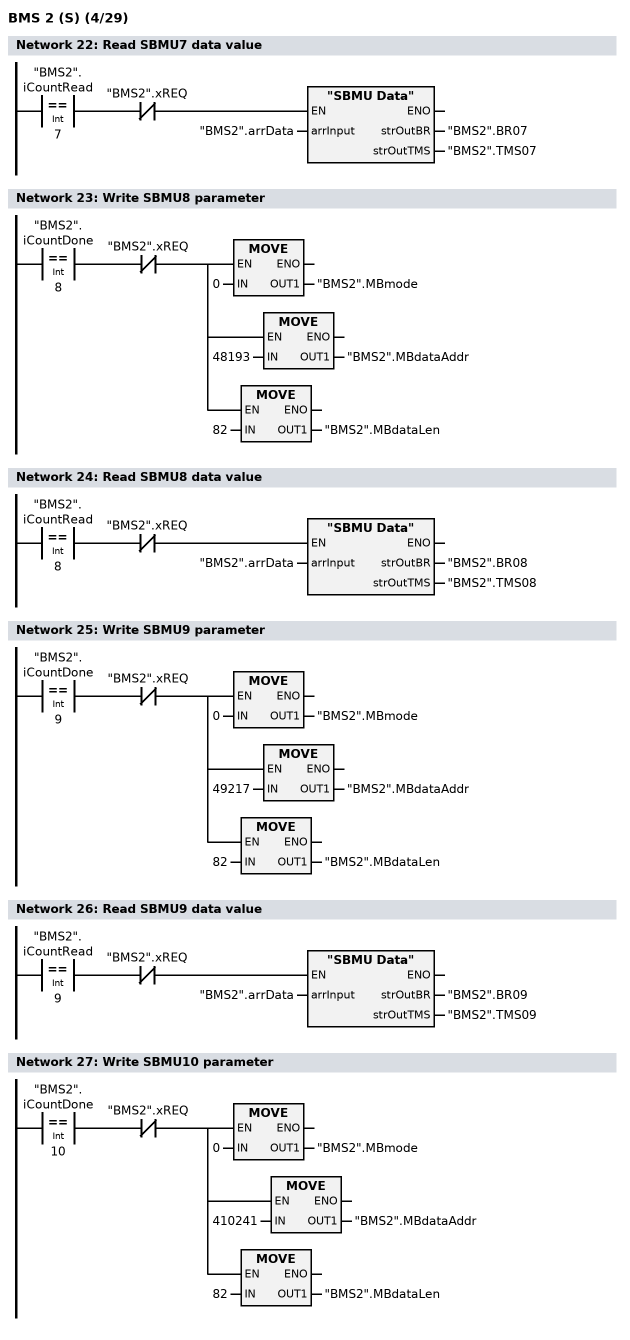
   RUNG wire#powerrail
      { S7_Templates := "SrcType := Int" } EQ_Contact(in1 := "BMS2".iCountRead, in2 := 7)
      I_Contact( "BMS2".xREQ )
      "SBMU Data"(arrInput := "BMS2".arrData, strOutBR => "BMS2".BR07, strOutTMS => "BMS2".TMS07)
   END_RUNG
   // the same network as SCL:
   IF ("BMS2".iCountRead = 7) AND NOT "BMS2".xREQ THEN
       "SBMU Data"(arrInput := "BMS2".arrData, strOutBR => "BMS2".BR07, strOutTMS => "BMS2".TMS07);
   END_IF;
END_REGION

REGION Network 23: Write SBMU8 parameter
   RUNG wire#powerrail
      { S7_Templates := "SrcType := Int" } EQ_Contact(in1 := "BMS2".iCountDone, in2 := 8)
      I_Contact( "BMS2".xREQ )
      wire#w1
      Move(in := 0, out1 => "BMS2".MBmode)
   END_RUNG
   RUNG wire#w1
      Move(in := 48193, out1 => "BMS2".MBdataAddr)
   END_RUNG
   RUNG wire#w1
      Move(in := 82, out1 => "BMS2".MBdataLen)
   END_RUNG
   // the same network as SCL:
   IF ("BMS2".iCountDone = 8) AND NOT "BMS2".xREQ THEN
       "BMS2".MBmode := 0;
       "BMS2".MBdataAddr := 48193;
       "BMS2".MBdataLen := 82;
   END_IF;
END_REGION

REGION Network 24: Read SBMU8 data value
   RUNG wire#powerrail
      { S7_Templates := "SrcType := Int" } EQ_Contact(in1 := "BMS2".iCountRead, in2 := 8)
      I_Contact( "BMS2".xREQ )
      "SBMU Data"(arrInput := "BMS2".arrData, strOutBR => "BMS2".BR08, strOutTMS => "BMS2".TMS08)
   END_RUNG
   // the same network as SCL:
   IF ("BMS2".iCountRead = 8) AND NOT "BMS2".xREQ THEN
       "SBMU Data"(arrInput := "BMS2".arrData, strOutBR => "BMS2".BR08, strOutTMS => "BMS2".TMS08);
   END_IF;
END_REGION

REGION Network 25: Write SBMU9 parameter
   RUNG wire#powerrail
      { S7_Templates := "SrcType := Int" } EQ_Contact(in1 := "BMS2".iCountDone, in2 := 9)
      I_Contact( "BMS2".xREQ )
      wire#w1
      Move(in := 0, out1 => "BMS2".MBmode)
   END_RUNG
   RUNG wire#w1
      Move(in := 49217, out1 => "BMS2".MBdataAddr)
   END_RUNG
   RUNG wire#w1
      Move(in := 82, out1 => "BMS2".MBdataLen)
   END_RUNG
   // the same network as SCL:
   IF ("BMS2".iCountDone = 9) AND NOT "BMS2".xREQ THEN
       "BMS2".MBmode := 0;
       "BMS2".MBdataAddr := 49217;
       "BMS2".MBdataLen := 82;
   END_IF;
END_REGION

REGION Network 26: Read SBMU9 data value
   RUNG wire#powerrail
      { S7_Templates := "SrcType := Int" } EQ_Contact(in1 := "BMS2".iCountRead, in2 := 9)
      I_Contact( "BMS2".xREQ )
      "SBMU Data"(arrInput := "BMS2".arrData, strOutBR => "BMS2".BR09, strOutTMS => "BMS2".TMS09)
   END_RUNG
   // the same network as SCL:
   IF ("BMS2".iCountRead = 9) AND NOT "BMS2".xREQ THEN
       "SBMU Data"(arrInput := "BMS2".arrData, strOutBR => "BMS2".BR09, strOutTMS => "BMS2".TMS09);
   END_IF;
END_REGION

REGION Network 27: Write SBMU10 parameter
   RUNG wire#powerrail
      { S7_Templates := "SrcType := Int" } EQ_Contact(in1 := "BMS2".iCountDone, in2 := 10)
      I_Contact( "BMS2".xREQ )
      wire#w1
      Move(in := 0, out1 => "BMS2".MBmode)
   END_RUNG
   RUNG wire#w1
      Move(in := 410241, out1 => "BMS2".MBdataAddr)
   END_RUNG
   RUNG wire#w1
      Move(in := 82, out1 => "BMS2".MBdataLen)
   END_RUNG
   // the same network as SCL:
   IF ("BMS2".iCountDone = 10) AND NOT "BMS2".xREQ THEN
       "BMS2".MBmode := 0;
       "BMS2".MBdataAddr := 410241;
       "BMS2".MBdataLen := 82;
   END_IF;
END_REGION

REGION Network 28: Read SBMU10 data value
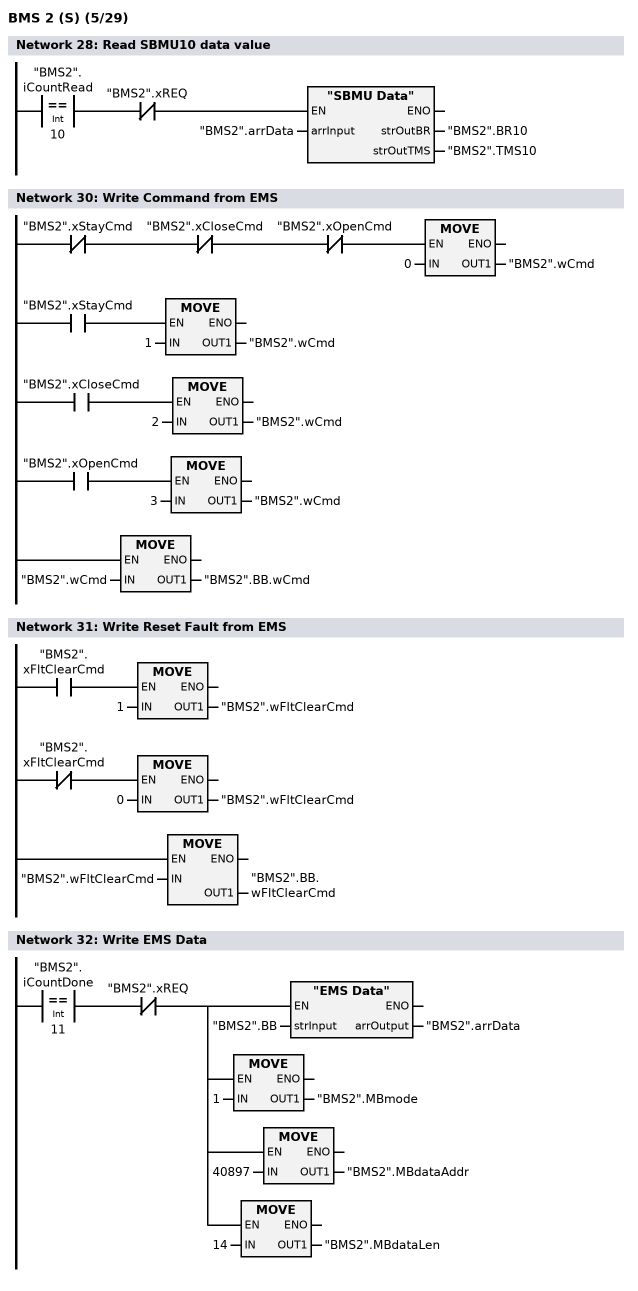
   RUNG wire#powerrail
      { S7_Templates := "SrcType := Int" } EQ_Contact(in1 := "BMS2".iCountRead, in2 := 10)
      I_Contact( "BMS2".xREQ )
      "SBMU Data"(arrInput := "BMS2".arrData, strOutBR => "BMS2".BR10, strOutTMS => "BMS2".TMS10)
   END_RUNG
   // the same network as SCL:
   IF ("BMS2".iCountRead = 10) AND NOT "BMS2".xREQ THEN
       "SBMU Data"(arrInput := "BMS2".arrData, strOutBR => "BMS2".BR10, strOutTMS => "BMS2".TMS10);
   END_IF;
END_REGION

REGION Network 30: Write Command from EMS
   RUNG wire#powerrail
      I_Contact( "BMS2".xStayCmd )
      I_Contact( "BMS2".xCloseCmd )
      I_Contact( "BMS2".xOpenCmd )
      Move(in := 0, out1 => "BMS2".wCmd)
   END_RUNG
   RUNG wire#powerrail
      Contact( "BMS2".xStayCmd )
      Move(in := 1, out1 => "BMS2".wCmd)
   END_RUNG
   RUNG wire#powerrail
      Contact( "BMS2".xCloseCmd )
      Move(in := 2, out1 => "BMS2".wCmd)
   END_RUNG
   RUNG wire#powerrail
      Contact( "BMS2".xOpenCmd )
      Move(in := 3, out1 => "BMS2".wCmd)
   END_RUNG
   RUNG wire#powerrail
      Move(in := "BMS2".wCmd, out1 => "BMS2".BB.wCmd)
   END_RUNG
   // the same network as SCL:
   IF NOT "BMS2".xStayCmd AND NOT "BMS2".xCloseCmd AND NOT "BMS2".xOpenCmd THEN "BMS2".wCmd := 0; END_IF;
   IF "BMS2".xStayCmd THEN "BMS2".wCmd := 1; END_IF;
   IF "BMS2".xCloseCmd THEN "BMS2".wCmd := 2; END_IF;
   IF "BMS2".xOpenCmd THEN "BMS2".wCmd := 3; END_IF;
   "BMS2".BB.wCmd := "BMS2".wCmd;
END_REGION

REGION Network 31: Write Reset Fault from EMS
   RUNG wire#powerrail
      Contact( "BMS2".xFltClearCmd )
      Move(in := 1, out1 => "BMS2".wFltClearCmd)
   END_RUNG
   RUNG wire#powerrail
      I_Contact( "BMS2".xFltClearCmd )
      Move(in := 0, out1 => "BMS2".wFltClearCmd)
   END_RUNG
   RUNG wire#powerrail
      Move(in := "BMS2".wFltClearCmd, out1 => "BMS2".BB.wFltClearCmd)
   END_RUNG
   // the same network as SCL:
   IF "BMS2".xFltClearCmd THEN "BMS2".wFltClearCmd := 1; END_IF;
   IF NOT "BMS2".xFltClearCmd THEN "BMS2".wFltClearCmd := 0; END_IF;
   "BMS2".BB.wFltClearCmd := "BMS2".wFltClearCmd;
END_REGION

REGION Network 32: Write EMS Data
   RUNG wire#powerrail
      { S7_Templates := "SrcType := Int" } EQ_Contact(in1 := "BMS2".iCountDone, in2 := 11)
      I_Contact( "BMS2".xREQ )
      wire#w1
      "EMS Data"(strInput := "BMS2".BB, arrOutput => "BMS2".arrData)
   END_RUNG
   RUNG wire#w1
      Move(in := 1, out1 => "BMS2".MBmode)
   END_RUNG
   RUNG wire#w1
      Move(in := 40897, out1 => "BMS2".MBdataAddr)
   END_RUNG
   RUNG wire#w1
      Move(in := 14, out1 => "BMS2".MBdataLen)
   END_RUNG
   // the same network as SCL:
   #_w1 := ("BMS2".iCountDone = 11) AND NOT "BMS2".xREQ;
   IF #_w1 THEN
       "EMS Data"(strInput := "BMS2".BB, arrOutput => "BMS2".arrData);
       "BMS2".MBmode := 1;
       "BMS2".MBdataAddr := 40897;
       "BMS2".MBdataLen := 14;
   END_IF;
END_REGION

REGION Network 34: Fault Modbus Communication
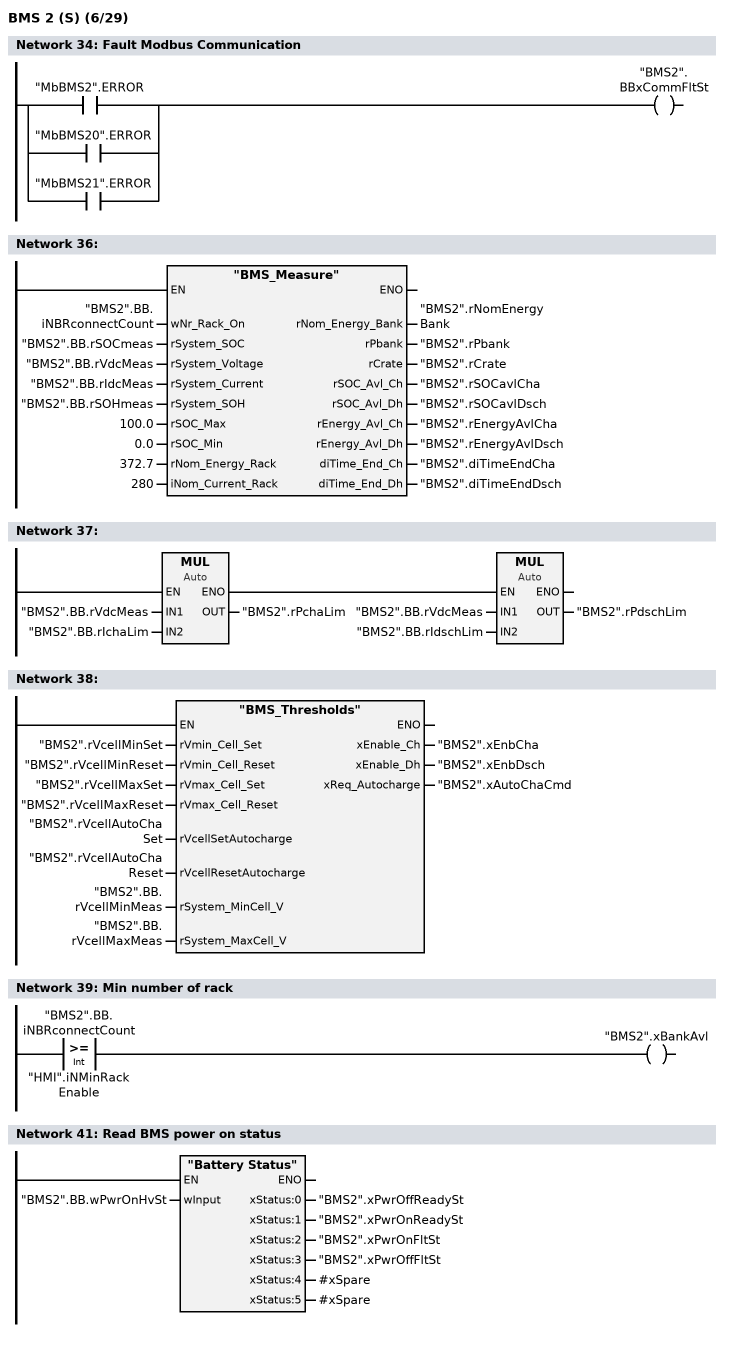
   RUNG wire#powerrail
      Contact( "MbBMS2".ERROR )
      wire#w1
      Coil( "BMS2".BBxCommFltSt )
   END_RUNG
   RUNG wire#powerrail
      Contact( "MbBMS20".ERROR )
   END_RUNG wire#w1
   RUNG wire#powerrail
      Contact( "MbBMS21".ERROR )
   END_RUNG wire#w1
   // the same network as SCL:
   "BMS2".BBxCommFltSt := "MbBMS2".ERROR OR "MbBMS20".ERROR OR "MbBMS21".ERROR;
END_REGION

REGION Network 36
   RUNG wire#powerrail
      "BMS_Measure"(wNr_Rack_On := "BMS2".BB.iNBRconnectCount, rSystem_SOC := "BMS2".BB.rSOCmeas, rSystem_Voltage := "BMS2".BB.rVdcMeas, rSystem_Current := "BMS2".BB.rIdcMeas, rSystem_SOH := "BMS2".BB.rSOHmeas, rSOC_Max := 100.0, rSOC_Min := 0.0, rNom_Energy_Rack := 372.7, iNom_Current_Rack := 280, rNom_Energy_Bank => "BMS2".rNomEnergyBank, rPbank => "BMS2".rPbank, rCrate => "BMS2".rCrate, rSOC_Avl_Ch => "BMS2".rSOCavlCha, rSOC_Avl_Dh => "BMS2".rSOCavlDsch, rEnergy_Avl_Ch => "BMS2".rEnergyAvlCha, rEnergy_Avl_Dh => "BMS2".rEnergyAvlDsch, diTime_End_Ch => "BMS2".diTimeEndCha, diTime_End_Dh => "BMS2".diTimeEndDsch)
   END_RUNG
   // the same network as SCL:
   "BMS_Measure"(wNr_Rack_On := "BMS2".BB.iNBRconnectCount,
                 rSystem_SOC := "BMS2".BB.rSOCmeas,
                 rSystem_Voltage := "BMS2".BB.rVdcMeas,
                 rSystem_Current := "BMS2".BB.rIdcMeas,
                 rSystem_SOH := "BMS2".BB.rSOHmeas,
                 rSOC_Max := 100.0,
                 rSOC_Min := 0.0,
                 rNom_Energy_Rack := 372.7,
                 iNom_Current_Rack := 280,
                 rNom_Energy_Bank => "BMS2".rNomEnergyBank,
                 rPbank => "BMS2".rPbank,
                 rCrate => "BMS2".rCrate,
                 rSOC_Avl_Ch => "BMS2".rSOCavlCha,
                 rSOC_Avl_Dh => "BMS2".rSOCavlDsch,
                 rEnergy_Avl_Ch => "BMS2".rEnergyAvlCha,
                 rEnergy_Avl_Dh => "BMS2".rEnergyAvlDsch,
                 diTime_End_Ch => "BMS2".diTimeEndCha,
                 diTime_End_Dh => "BMS2".diTimeEndDsch);
END_REGION

REGION Network 37
   RUNG wire#powerrail
      Mul(in1 := "BMS2".BB.rVdcMeas, in2 := "BMS2".BB.rIchaLim, out => "BMS2".rPchaLim)
      Mul(in1 := "BMS2".BB.rVdcMeas, in2 := "BMS2".BB.rIdschLim, out => "BMS2".rPdschLim)
   END_RUNG
   // the same network as SCL:
   "BMS2".rPchaLim := "BMS2".BB.rVdcMeas * "BMS2".BB.rIchaLim;
   "BMS2".rPdschLim := "BMS2".BB.rVdcMeas * "BMS2".BB.rIdschLim;
END_REGION

REGION Network 38
   RUNG wire#powerrail
      "BMS_Thresholds"(rVmin_Cell_Set := "BMS2".rVcellMinSet, rVmin_Cell_Reset := "BMS2".rVcellMinReset, rVmax_Cell_Set := "BMS2".rVcellMaxSet, rVmax_Cell_Reset := "BMS2".rVcellMaxReset, rVcellSetAutocharge := "BMS2".rVcellAutoChaSet, rVcellResetAutocharge := "BMS2".rVcellAutoChaReset, rSystem_MinCell_V := "BMS2".BB.rVcellMinMeas, rSystem_MaxCell_V := "BMS2".BB.rVcellMaxMeas, xEnable_Ch => "BMS2".xEnbCha, xEnable_Dh => "BMS2".xEnbDsch, xReq_Autocharge => "BMS2".xAutoChaCmd)
   END_RUNG
   // the same network as SCL:
   "BMS_Thresholds"(rVmin_Cell_Set := "BMS2".rVcellMinSet,
                    rVmin_Cell_Reset := "BMS2".rVcellMinReset,
                    rVmax_Cell_Set := "BMS2".rVcellMaxSet,
                    rVmax_Cell_Reset := "BMS2".rVcellMaxReset,
                    rVcellSetAutocharge := "BMS2".rVcellAutoChaSet,
                    rVcellResetAutocharge := "BMS2".rVcellAutoChaReset,
                    rSystem_MinCell_V := "BMS2".BB.rVcellMinMeas,
                    rSystem_MaxCell_V := "BMS2".BB.rVcellMaxMeas,
                    xEnable_Ch => "BMS2".xEnbCha,
                    xEnable_Dh => "BMS2".xEnbDsch,
                    xReq_Autocharge => "BMS2".xAutoChaCmd);
END_REGION

REGION Network 39: Min number of rack
   RUNG wire#powerrail
      { S7_Templates := "SrcType := Int" } GE_Contact(in1 := "BMS2".BB.iNBRconnectCount, in2 := "HMI".iNMinRackEnable)
      Coil( "BMS2".xBankAvl )
   END_RUNG
   // the same network as SCL:
   "BMS2".xBankAvl := "BMS2".BB.iNBRconnectCount >= "HMI".iNMinRackEnable;
END_REGION

REGION Network 41: Read BMS power on status
   RUNG wire#powerrail
      "Battery Status"(wInput := "BMS2".BB.wPwrOnHvSt, "xStatus:0" => "BMS2".xPwrOffReadySt, "xStatus:1" => "BMS2".xPwrOnReadySt, "xStatus:2" => "BMS2".xPwrOnFltSt, "xStatus:3" => "BMS2".xPwrOffFltSt, "xStatus:4" => #xSpare, "xStatus:5" => #xSpare)
   END_RUNG
   // the same network as SCL:
   "Battery Status"(wInput := "BMS2".BB.wPwrOnHvSt,
                    "xStatus:0" => "BMS2".xPwrOffReadySt,
                    "xStatus:1" => "BMS2".xPwrOnReadySt,
                    "xStatus:2" => "BMS2".xPwrOnFltSt,
                    "xStatus:3" => "BMS2".xPwrOffFltSt,
                    "xStatus:4" => #xSpare,
                    "xStatus:5" => #xSpare);
END_REGION

REGION Network 42: Read BMS status
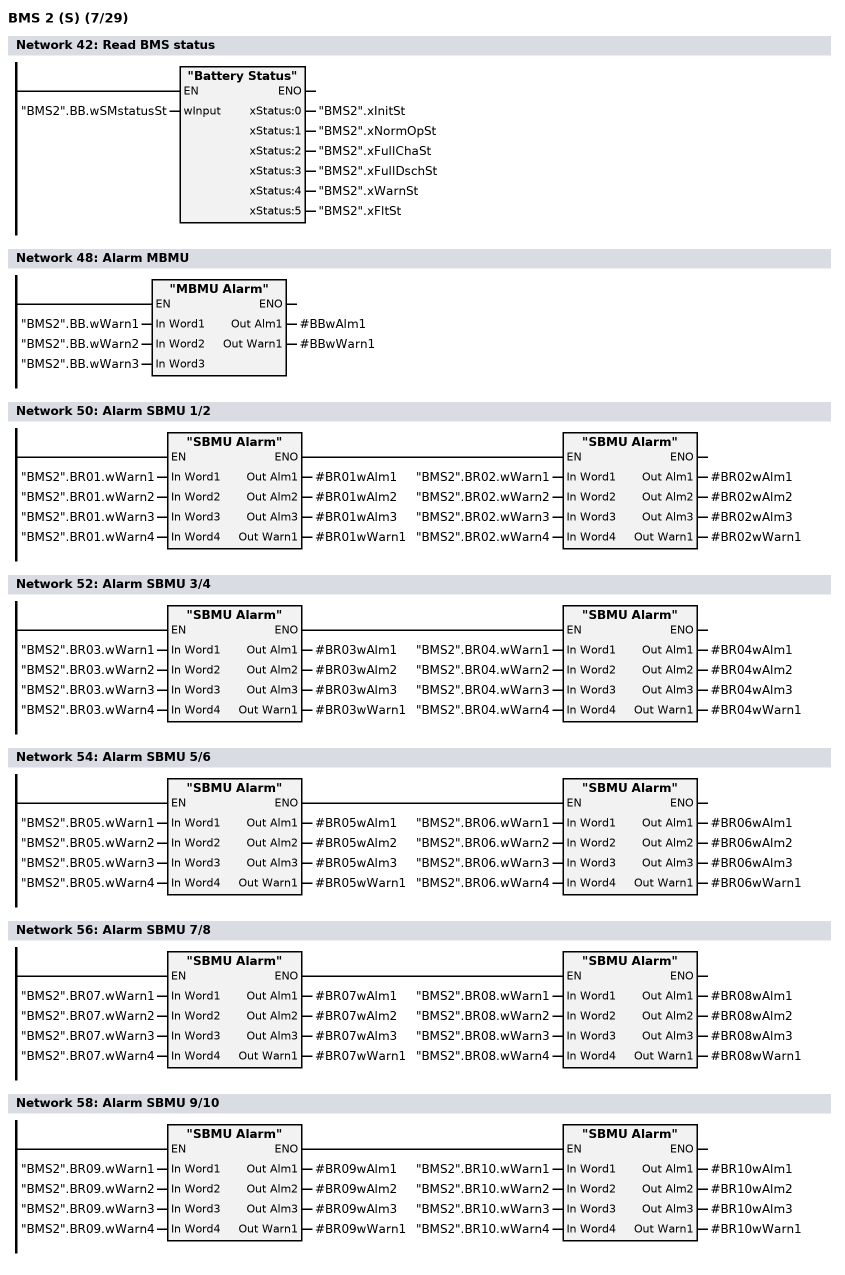
   RUNG wire#powerrail
      "Battery Status"(wInput := "BMS2".BB.wSMstatusSt, "xStatus:0" => "BMS2".xInitSt, "xStatus:1" => "BMS2".xNormOpSt, "xStatus:2" => "BMS2".xFullChaSt, "xStatus:3" => "BMS2".xFullDschSt, "xStatus:4" => "BMS2".xWarnSt, "xStatus:5" => "BMS2".xFltSt)
   END_RUNG
   // the same network as SCL:
   "Battery Status"(wInput := "BMS2".BB.wSMstatusSt,
                    "xStatus:0" => "BMS2".xInitSt,
                    "xStatus:1" => "BMS2".xNormOpSt,
                    "xStatus:2" => "BMS2".xFullChaSt,
                    "xStatus:3" => "BMS2".xFullDschSt,
                    "xStatus:4" => "BMS2".xWarnSt,
                    "xStatus:5" => "BMS2".xFltSt);
END_REGION

REGION Network 44 (SCL): Rack Fault Status
   "BMS2".wRackFlt.%X0 := "BMS2".BR01xFltSt;
   "BMS2".wRackFlt.%X1 := "BMS2".BR02xFltSt;
   "BMS2".wRackFlt.%X2 := "BMS2".BR03xFltSt;
   "BMS2".wRackFlt.%X3 := "BMS2".BR04xFltSt;
   "BMS2".wRackFlt.%X4 := "BMS2".BR05xFltSt;
   "BMS2".wRackFlt.%X5 := "BMS2".BR06xFltSt;
   "BMS2".wRackFlt.%X6 := "BMS2".BR07xFltSt;
   "BMS2".wRackFlt.%X7 := "BMS2".BR08xFltSt;
   "BMS2".wRackFlt.%X8 := "BMS2".BR09xFltSt;
   "BMS2".wRackFlt.%X9 := "BMS2".BR10xFltSt;
END_REGION

REGION Network 45 (SCL): Rack On Status
   "BMS2".wRackOn.%X0 := "BMS2".BR01.xKposSt;
   "BMS2".wRackOn.%X1 := "BMS2".BR02.xKposSt;
   "BMS2".wRackOn.%X2 := "BMS2".BR03.xKposSt;
   "BMS2".wRackOn.%X3 := "BMS2".BR04.xKposSt;
   "BMS2".wRackOn.%X4 := "BMS2".BR05.xKposSt;
   "BMS2".wRackOn.%X5 := "BMS2".BR06.xKposSt;
   "BMS2".wRackOn.%X6 := "BMS2".BR07.xKposSt;
   "BMS2".wRackOn.%X7 := "BMS2".BR08.xKposSt;
   "BMS2".wRackOn.%X8 := "BMS2".BR09.xKposSt;
   "BMS2".wRackOn.%X9 := "BMS2".BR10.xKposSt;
END_REGION

REGION Network 46 (SCL): Status Switch Gear
   IF
       NOT "BMS2".BR01wAlm2.%X12 OR
       NOT "BMS2".BR02wAlm2.%X12 OR
       NOT "BMS2".BR03wAlm2.%X12 OR
       NOT "BMS2".BR04wAlm2.%X12 OR
       NOT "BMS2".BR05wAlm2.%X12 OR
       NOT "BMS2".BR06wAlm2.%X12 OR
       NOT "BMS2".BR07wAlm2.%X12 OR
       NOT "BMS2".BR08wAlm2.%X12 OR
       NOT "BMS2".BR09wAlm2.%X12 OR
       NOT "BMS2".BR10wAlm2.%X12 THEN

       "BMS2".xSwitchGearSt := True;
   ELSE
       "BMS2".xSwitchGearSt := False;
   END_IF;
END_REGION

REGION Network 48: Alarm MBMU
   RUNG wire#powerrail
      "MBMU Alarm"("In Word1" := "BMS2".BB.wWarn1, "In Word2" := "BMS2".BB.wWarn2, "In Word3" := "BMS2".BB.wWarn3, "Out Alm1" => #BBwAlm1, "Out Warn1" => #BBwWarn1)
   END_RUNG
   // the same network as SCL:
   "MBMU Alarm"("In Word1" := "BMS2".BB.wWarn1,
                "In Word2" := "BMS2".BB.wWarn2,
                "In Word3" := "BMS2".BB.wWarn3,
                "Out Alm1" => #BBwAlm1,
                "Out Warn1" => #BBwWarn1);
END_REGION

REGION Network 49 (SCL): Alarm MBMU to HMI
   IF "HMI".xBB2AlmDisable OR"HMI".xPEMSAlmDisable OR"HMI".xPIAlmDisable
   THEN
       "BMS2".BBwAlm1 := 0;
       "BMS2".BBwWarn1 := 0;
   ELSE
       "BMS2".BBwAlm1 := #BBwAlm1;
       "BMS2".BBwWarn1 := #BBwWarn1;
   END_IF;
END_REGION

REGION Network 50: Alarm SBMU 1/2
   RUNG wire#powerrail
      "SBMU Alarm"("In Word1" := "BMS2".BR01.wWarn1, "In Word2" := "BMS2".BR01.wWarn2, "In Word3" := "BMS2".BR01.wWarn3, "In Word4" := "BMS2".BR01.wWarn4, "Out Alm1" => #BR01wAlm1, "Out Alm2" => #BR01wAlm2, "Out Alm3" => #BR01wAlm3, "Out Warn1" => #BR01wWarn1)
      "SBMU Alarm"("In Word1" := "BMS2".BR02.wWarn1, "In Word2" := "BMS2".BR02.wWarn2, "In Word3" := "BMS2".BR02.wWarn3, "In Word4" := "BMS2".BR02.wWarn4, "Out Alm1" => #BR02wAlm1, "Out Alm2" => #BR02wAlm2, "Out Alm3" => #BR02wAlm3, "Out Warn1" => #BR02wWarn1)
   END_RUNG
   // the same network as SCL:
   "SBMU Alarm"("In Word1" := "BMS2".BR01.wWarn1,
                "In Word2" := "BMS2".BR01.wWarn2,
                "In Word3" := "BMS2".BR01.wWarn3,
                "In Word4" := "BMS2".BR01.wWarn4,
                "Out Alm1" => #BR01wAlm1,
                "Out Alm2" => #BR01wAlm2,
                "Out Alm3" => #BR01wAlm3,
                "Out Warn1" => #BR01wWarn1,
                ENO => #_w1);
   IF #_w1 THEN
       "SBMU Alarm"("In Word1" := "BMS2".BR02.wWarn1,
                    "In Word2" := "BMS2".BR02.wWarn2,
                    "In Word3" := "BMS2".BR02.wWarn3,
                    "In Word4" := "BMS2".BR02.wWarn4,
                    "Out Alm1" => #BR02wAlm1,
                    "Out Alm2" => #BR02wAlm2,
                    "Out Alm3" => #BR02wAlm3,
                    "Out Warn1" => #BR02wWarn1);
   END_IF;
END_REGION

REGION Network 51 (SCL): Alarm SBMU 1/2 to HMI
   IF "HMI".xBB2BR1AlmDisable OR "HMI".xBB2AlmDisable OR "HMI".xPEMSAlmDisable OR "HMI".xPIAlmDisable
   THEN
       "BMS2".BR01wAlm1 := 0;
       "BMS2".BR01wAlm2 := 0;
       "BMS2".BR01wAlm3 := 0;
       "BMS2".BR01wWarn1 := 0;
   ELSE
       "BMS2".BR01wAlm1 := #BR01wAlm1;
       "BMS2".BR01wAlm2 := #BR01wAlm2;
       "BMS2".BR01wAlm3 := #BR01wAlm3;
       "BMS2".BR01wWarn1 := #BR01wWarn1;
   END_IF;

   IF "HMI".xBB2BR2AlmDisable OR "HMI".xBB2AlmDisable OR "HMI".xPEMSAlmDisable OR "HMI".xPIAlmDisable
   THEN
       "BMS2".BR02wAlm1 := 0;
       "BMS2".BR02wAlm2 := 0;
       "BMS2".BR02wAlm3 := 0;
       "BMS2".BR02wWarn1 := 0;
   ELSE
       "BMS2".BR02wAlm1 := #BR02wAlm1;
       "BMS2".BR02wAlm2 := #BR02wAlm2;
       "BMS2".BR02wAlm3 := #BR02wAlm3;
       "BMS2".BR02wWarn1 := #BR02wWarn1;
   END_IF;
END_REGION

REGION Network 52: Alarm SBMU 3/4
   RUNG wire#powerrail
      "SBMU Alarm"("In Word1" := "BMS2".BR03.wWarn1, "In Word2" := "BMS2".BR03.wWarn2, "In Word3" := "BMS2".BR03.wWarn3, "In Word4" := "BMS2".BR03.wWarn4, "Out Alm1" => #BR03wAlm1, "Out Alm2" => #BR03wAlm2, "Out Alm3" => #BR03wAlm3, "Out Warn1" => #BR03wWarn1)
      "SBMU Alarm"("In Word1" := "BMS2".BR04.wWarn1, "In Word2" := "BMS2".BR04.wWarn2, "In Word3" := "BMS2".BR04.wWarn3, "In Word4" := "BMS2".BR04.wWarn4, "Out Alm1" => #BR04wAlm1, "Out Alm2" => #BR04wAlm2, "Out Alm3" => #BR04wAlm3, "Out Warn1" => #BR04wWarn1)
   END_RUNG
   // the same network as SCL:
   "SBMU Alarm"("In Word1" := "BMS2".BR03.wWarn1,
                "In Word2" := "BMS2".BR03.wWarn2,
                "In Word3" := "BMS2".BR03.wWarn3,
                "In Word4" := "BMS2".BR03.wWarn4,
                "Out Alm1" => #BR03wAlm1,
                "Out Alm2" => #BR03wAlm2,
                "Out Alm3" => #BR03wAlm3,
                "Out Warn1" => #BR03wWarn1,
                ENO => #_w1);
   IF #_w1 THEN
       "SBMU Alarm"("In Word1" := "BMS2".BR04.wWarn1,
                    "In Word2" := "BMS2".BR04.wWarn2,
                    "In Word3" := "BMS2".BR04.wWarn3,
                    "In Word4" := "BMS2".BR04.wWarn4,
                    "Out Alm1" => #BR04wAlm1,
                    "Out Alm2" => #BR04wAlm2,
                    "Out Alm3" => #BR04wAlm3,
                    "Out Warn1" => #BR04wWarn1);
   END_IF;
END_REGION

REGION Network 53 (SCL): Alarm SBMU 3/4 to HMI
   IF "HMI".xBB2BR3AlmDisable OR "HMI".xBB2AlmDisable OR "HMI".xPEMSAlmDisable OR "HMI".xPIAlmDisable
   THEN
       "BMS2".BR03wAlm1 := 0;
       "BMS2".BR03wAlm2 := 0;
       "BMS2".BR03wAlm3 := 0;
       "BMS2".BR03wWarn1 := 0;
   ELSE
       "BMS2".BR03wAlm1 := #BR03wAlm1;
       "BMS2".BR03wAlm2 := #BR03wAlm2;
       "BMS2".BR03wAlm3 := #BR03wAlm3;
       "BMS2".BR03wWarn1 := #BR03wWarn1;
   END_IF;

   IF "HMI".xBB2BR4AlmDisable OR "HMI".xBB2AlmDisable OR "HMI".xPEMSAlmDisable OR "HMI".xPIAlmDisable
   THEN
       "BMS2".BR04wAlm1 := 0;
       "BMS2".BR04wAlm2 := 0;
       "BMS2".BR04wAlm3 := 0;
       "BMS2".BR04wWarn1 := 0;
   ELSE
       "BMS2".BR04wAlm1 := #BR04wAlm1;
       "BMS2".BR04wAlm2 := #BR04wAlm2;
       "BMS2".BR04wAlm3 := #BR04wAlm3;
       "BMS2".BR04wWarn1 := #BR04wWarn1;
   END_IF;
END_REGION

REGION Network 54: Alarm SBMU 5/6
   RUNG wire#powerrail
      "SBMU Alarm"("In Word1" := "BMS2".BR05.wWarn1, "In Word2" := "BMS2".BR05.wWarn2, "In Word3" := "BMS2".BR05.wWarn3, "In Word4" := "BMS2".BR05.wWarn4, "Out Alm1" => #BR05wAlm1, "Out Alm2" => #BR05wAlm2, "Out Alm3" => #BR05wAlm3, "Out Warn1" => #BR05wWarn1)
      "SBMU Alarm"("In Word1" := "BMS2".BR06.wWarn1, "In Word2" := "BMS2".BR06.wWarn2, "In Word3" := "BMS2".BR06.wWarn3, "In Word4" := "BMS2".BR06.wWarn4, "Out Alm1" => #BR06wAlm1, "Out Alm2" => #BR06wAlm2, "Out Alm3" => #BR06wAlm3, "Out Warn1" => #BR06wWarn1)
   END_RUNG
   // the same network as SCL:
   "SBMU Alarm"("In Word1" := "BMS2".BR05.wWarn1,
                "In Word2" := "BMS2".BR05.wWarn2,
                "In Word3" := "BMS2".BR05.wWarn3,
                "In Word4" := "BMS2".BR05.wWarn4,
                "Out Alm1" => #BR05wAlm1,
                "Out Alm2" => #BR05wAlm2,
                "Out Alm3" => #BR05wAlm3,
                "Out Warn1" => #BR05wWarn1,
                ENO => #_w1);
   IF #_w1 THEN
       "SBMU Alarm"("In Word1" := "BMS2".BR06.wWarn1,
                    "In Word2" := "BMS2".BR06.wWarn2,
                    "In Word3" := "BMS2".BR06.wWarn3,
                    "In Word4" := "BMS2".BR06.wWarn4,
                    "Out Alm1" => #BR06wAlm1,
                    "Out Alm2" => #BR06wAlm2,
                    "Out Alm3" => #BR06wAlm3,
                    "Out Warn1" => #BR06wWarn1);
   END_IF;
END_REGION

REGION Network 55 (SCL): Alarm SBMU 5/6 to HMI
   IF "HMI".xBB2BR5AlmDisable OR "HMI".xBB2AlmDisable OR "HMI".xPEMSAlmDisable OR "HMI".xPIAlmDisable
   THEN
       "BMS2".BR05wAlm1 := 0;
       "BMS2".BR05wAlm2 := 0;
       "BMS2".BR05wAlm3 := 0;
       "BMS2".BR05wWarn1 := 0;
   ELSE
       "BMS2".BR05wAlm1 := #BR05wAlm1;
       "BMS2".BR05wAlm2 := #BR05wAlm2;
       "BMS2".BR05wAlm3 := #BR05wAlm3;
       "BMS2".BR05wWarn1 := #BR05wWarn1;
   END_IF;

   IF "HMI".xBB2BR6AlmDisable OR "HMI".xBB2AlmDisable OR "HMI".xPEMSAlmDisable OR "HMI".xPIAlmDisable
   THEN
       "BMS2".BR06wAlm1 := 0;
       "BMS2".BR06wAlm2 := 0;
       "BMS2".BR06wAlm3 := 0;
       "BMS2".BR06wWarn1 := 0;
   ELSE
       "BMS2".BR06wAlm1 := #BR06wAlm1;
       "BMS2".BR06wAlm2 := #BR06wAlm2;
       "BMS2".BR06wAlm3 := #BR06wAlm3;
       "BMS2".BR06wWarn1 := #BR06wWarn1;
   END_IF;
END_REGION

REGION Network 56: Alarm SBMU 7/8
   RUNG wire#powerrail
      "SBMU Alarm"("In Word1" := "BMS2".BR07.wWarn1, "In Word2" := "BMS2".BR07.wWarn2, "In Word3" := "BMS2".BR07.wWarn3, "In Word4" := "BMS2".BR07.wWarn4, "Out Alm1" => #BR07wAlm1, "Out Alm2" => #BR07wAlm2, "Out Alm3" => #BR07wAlm3, "Out Warn1" => #BR07wWarn1)
      "SBMU Alarm"("In Word1" := "BMS2".BR08.wWarn1, "In Word2" := "BMS2".BR08.wWarn2, "In Word3" := "BMS2".BR08.wWarn3, "In Word4" := "BMS2".BR08.wWarn4, "Out Alm1" => #BR08wAlm1, "Out Alm2" => #BR08wAlm2, "Out Alm3" => #BR08wAlm3, "Out Warn1" => #BR08wWarn1)
   END_RUNG
   // the same network as SCL:
   "SBMU Alarm"("In Word1" := "BMS2".BR07.wWarn1,
                "In Word2" := "BMS2".BR07.wWarn2,
                "In Word3" := "BMS2".BR07.wWarn3,
                "In Word4" := "BMS2".BR07.wWarn4,
                "Out Alm1" => #BR07wAlm1,
                "Out Alm2" => #BR07wAlm2,
                "Out Alm3" => #BR07wAlm3,
                "Out Warn1" => #BR07wWarn1,
                ENO => #_w1);
   IF #_w1 THEN
       "SBMU Alarm"("In Word1" := "BMS2".BR08.wWarn1,
                    "In Word2" := "BMS2".BR08.wWarn2,
                    "In Word3" := "BMS2".BR08.wWarn3,
                    "In Word4" := "BMS2".BR08.wWarn4,
                    "Out Alm1" => #BR08wAlm1,
                    "Out Alm2" => #BR08wAlm2,
                    "Out Alm3" => #BR08wAlm3,
                    "Out Warn1" => #BR08wWarn1);
   END_IF;
END_REGION

REGION Network 57 (SCL): Alarm SBMU 7/8 to HMI
   IF "HMI".xBB2BR7AlmDisable OR "HMI".xBB2AlmDisable OR "HMI".xPEMSAlmDisable OR "HMI".xPIAlmDisable
   THEN
       "BMS2".BR07wAlm1 := 0;
       "BMS2".BR07wAlm2 := 0;
       "BMS2".BR07wAlm3 := 0;
       "BMS2".BR07wWarn1 := 0;
   ELSE
       "BMS2".BR07wAlm1 := #BR07wAlm1;
       "BMS2".BR07wAlm2 := #BR07wAlm2;
       "BMS2".BR07wAlm3 := #BR07wAlm3;
       "BMS2".BR07wWarn1 := #BR07wWarn1;
   END_IF;

   IF "HMI".xBB2BR8AlmDisable OR "HMI".xBB2AlmDisable OR "HMI".xPEMSAlmDisable OR "HMI".xPIAlmDisable
   THEN
       "BMS2".BR08wAlm1 := 0;
       "BMS2".BR08wAlm2 := 0;
       "BMS2".BR08wAlm3 := 0;
       "BMS2".BR08wWarn1 := 0;
   ELSE
       "BMS2".BR08wAlm1 := #BR08wAlm1;
       "BMS2".BR08wAlm2 := #BR08wAlm2;
       "BMS2".BR08wAlm3 := #BR08wAlm3;
       "BMS2".BR08wWarn1 := #BR08wWarn1;
   END_IF;
END_REGION

REGION Network 58: Alarm SBMU 9/10
   RUNG wire#powerrail
      "SBMU Alarm"("In Word1" := "BMS2".BR09.wWarn1, "In Word2" := "BMS2".BR09.wWarn2, "In Word3" := "BMS2".BR09.wWarn3, "In Word4" := "BMS2".BR09.wWarn4, "Out Alm1" => #BR09wAlm1, "Out Alm2" => #BR09wAlm2, "Out Alm3" => #BR09wAlm3, "Out Warn1" => #BR09wWarn1)
      "SBMU Alarm"("In Word1" := "BMS2".BR10.wWarn1, "In Word2" := "BMS2".BR10.wWarn2, "In Word3" := "BMS2".BR10.wWarn3, "In Word4" := "BMS2".BR10.wWarn4, "Out Alm1" => #BR10wAlm1, "Out Alm2" => #BR10wAlm2, "Out Alm3" => #BR10wAlm3, "Out Warn1" => #BR10wWarn1)
   END_RUNG
   // the same network as SCL:
   "SBMU Alarm"("In Word1" := "BMS2".BR09.wWarn1,
                "In Word2" := "BMS2".BR09.wWarn2,
                "In Word3" := "BMS2".BR09.wWarn3,
                "In Word4" := "BMS2".BR09.wWarn4,
                "Out Alm1" => #BR09wAlm1,
                "Out Alm2" => #BR09wAlm2,
                "Out Alm3" => #BR09wAlm3,
                "Out Warn1" => #BR09wWarn1,
                ENO => #_w1);
   IF #_w1 THEN
       "SBMU Alarm"("In Word1" := "BMS2".BR10.wWarn1,
                    "In Word2" := "BMS2".BR10.wWarn2,
                    "In Word3" := "BMS2".BR10.wWarn3,
                    "In Word4" := "BMS2".BR10.wWarn4,
                    "Out Alm1" => #BR10wAlm1,
                    "Out Alm2" => #BR10wAlm2,
                    "Out Alm3" => #BR10wAlm3,
                    "Out Warn1" => #BR10wWarn1);
   END_IF;
END_REGION

REGION Network 59 (SCL): Alarm SBMU 9/10 to HMI
   IF "HMI".xBB2BR9AlmDisable OR "HMI".xBB2AlmDisable OR "HMI".xPEMSAlmDisable OR "HMI".xPIAlmDisable
   THEN
       "BMS2".BR09wAlm1 := 0;
       "BMS2".BR09wAlm2 := 0;
       "BMS2".BR09wAlm3 := 0;
       "BMS2".BR09wWarn1 := 0;
   ELSE
       "BMS2".BR09wAlm1 := #BR09wAlm1;
       "BMS2".BR09wAlm2 := #BR09wAlm2;
       "BMS2".BR09wAlm3 := #BR09wAlm3;
       "BMS2".BR09wWarn1 := #BR09wWarn1;
   END_IF;

   IF "HMI".xBB2BR10AlmDisable OR "HMI".xBB2AlmDisable OR "HMI".xPEMSAlmDisable OR "HMI".xPIAlmDisable
   THEN
       "BMS2".BR10wAlm1 := 0;
       "BMS2".BR10wAlm2 := 0;
       "BMS2".BR10wAlm3 := 0;
       "BMS2".BR10wWarn1 := 0;
   ELSE
       "BMS2".BR10wAlm1 := #BR10wAlm1;
       "BMS2".BR10wAlm2 := #BR10wAlm2;
       "BMS2".BR10wAlm3 := #BR10wAlm3;
       "BMS2".BR10wWarn1 := #BR10wWarn1;
   END_IF;
END_REGION

REGION Network 61: BMS2 Fault SubSystem
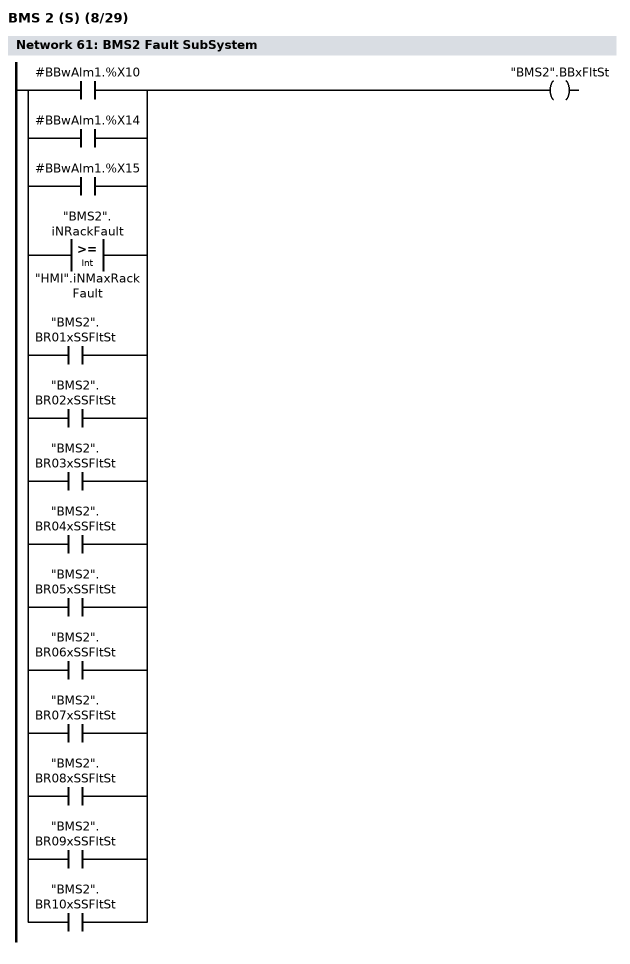
   RUNG wire#powerrail
      Contact( #BBwAlm1.%X10 )
      wire#w1
      Coil( "BMS2".BBxFltSt )
   END_RUNG
   RUNG wire#powerrail
      Contact( #BBwAlm1.%X14 )
   END_RUNG wire#w1
   RUNG wire#powerrail
      Contact( #BBwAlm1.%X15 )
   END_RUNG wire#w1
   RUNG wire#powerrail
      { S7_Templates := "SrcType := Int" } GE_Contact(in1 := "BMS2".iNRackFault, in2 := "HMI".iNMaxRackFault)
   END_RUNG wire#w1
   RUNG wire#powerrail
      Contact( "BMS2".BR01xSSFltSt )
   END_RUNG wire#w1
   RUNG wire#powerrail
      Contact( "BMS2".BR02xSSFltSt )
   END_RUNG wire#w1
   RUNG wire#powerrail
      Contact( "BMS2".BR03xSSFltSt )
   END_RUNG wire#w1
   RUNG wire#powerrail
      Contact( "BMS2".BR04xSSFltSt )
   END_RUNG wire#w1
   RUNG wire#powerrail
      Contact( "BMS2".BR05xSSFltSt )
   END_RUNG wire#w1
   RUNG wire#powerrail
      Contact( "BMS2".BR06xSSFltSt )
   END_RUNG wire#w1
   RUNG wire#powerrail
      Contact( "BMS2".BR07xSSFltSt )
   END_RUNG wire#w1
   RUNG wire#powerrail
      Contact( "BMS2".BR08xSSFltSt )
   END_RUNG wire#w1
   RUNG wire#powerrail
      Contact( "BMS2".BR09xSSFltSt )
   END_RUNG wire#w1
   RUNG wire#powerrail
      Contact( "BMS2".BR10xSSFltSt )
   END_RUNG wire#w1
   // the same network as SCL:
   "BMS2".BBxFltSt := #BBwAlm1.%X10 OR #BBwAlm1.%X14 OR #BBwAlm1.%X15 OR ("BMS2".iNRackFault >= "HMI".iNMaxRackFault) OR "BMS2".BR01xSSFltSt OR "BMS2".BR02xSSFltSt OR "BMS2".BR03xSSFltSt OR "BMS2".BR04xSSFltSt OR "BMS2".BR05xSSFltSt OR "BMS2".BR06xSSFltSt OR "BMS2".BR07xSSFltSt OR "BMS2".BR08xSSFltSt OR "BMS2".BR09xSSFltSt OR "BMS2".BR10xSSFltSt;
END_REGION

REGION Network 62: BMS2 Alarm
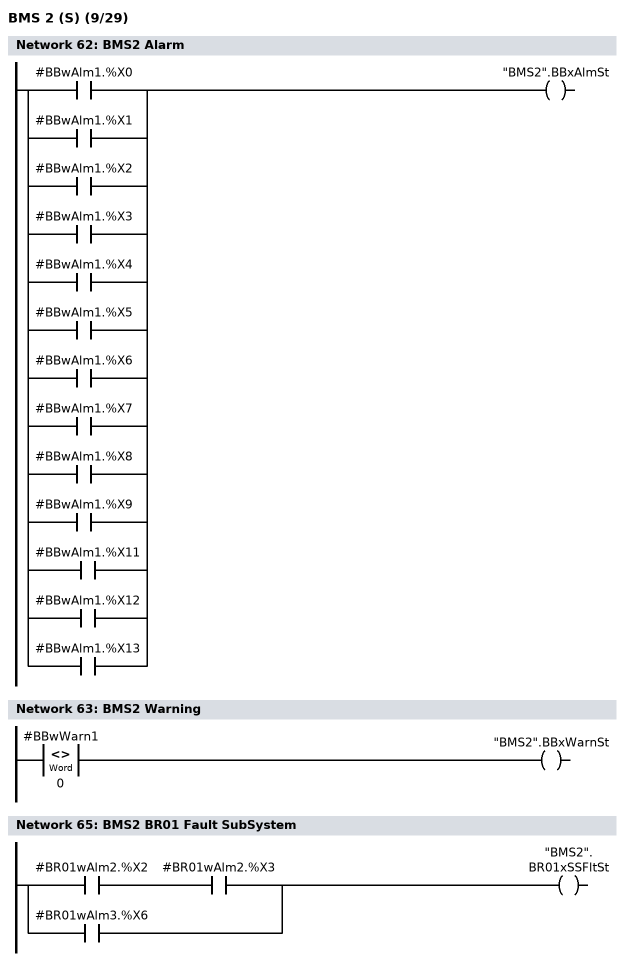
   RUNG wire#powerrail
      Contact( #BBwAlm1.%X0 )
      wire#w1
      Coil( "BMS2".BBxAlmSt )
   END_RUNG
   RUNG wire#powerrail
      Contact( #BBwAlm1.%X1 )
   END_RUNG wire#w1
   RUNG wire#powerrail
      Contact( #BBwAlm1.%X2 )
   END_RUNG wire#w1
   RUNG wire#powerrail
      Contact( #BBwAlm1.%X3 )
   END_RUNG wire#w1
   RUNG wire#powerrail
      Contact( #BBwAlm1.%X4 )
   END_RUNG wire#w1
   RUNG wire#powerrail
      Contact( #BBwAlm1.%X5 )
   END_RUNG wire#w1
   RUNG wire#powerrail
      Contact( #BBwAlm1.%X6 )
   END_RUNG wire#w1
   RUNG wire#powerrail
      Contact( #BBwAlm1.%X7 )
   END_RUNG wire#w1
   RUNG wire#powerrail
      Contact( #BBwAlm1.%X8 )
   END_RUNG wire#w1
   RUNG wire#powerrail
      Contact( #BBwAlm1.%X9 )
   END_RUNG wire#w1
   RUNG wire#powerrail
      Contact( #BBwAlm1.%X11 )
   END_RUNG wire#w1
   RUNG wire#powerrail
      Contact( #BBwAlm1.%X12 )
   END_RUNG wire#w1
   RUNG wire#powerrail
      Contact( #BBwAlm1.%X13 )
   END_RUNG wire#w1
   // the same network as SCL:
   "BMS2".BBxAlmSt := #BBwAlm1.%X0 OR #BBwAlm1.%X1 OR #BBwAlm1.%X2 OR #BBwAlm1.%X3 OR #BBwAlm1.%X4 OR #BBwAlm1.%X5 OR #BBwAlm1.%X6 OR #BBwAlm1.%X7 OR #BBwAlm1.%X8 OR #BBwAlm1.%X9 OR #BBwAlm1.%X11 OR #BBwAlm1.%X12 OR #BBwAlm1.%X13;
END_REGION

REGION Network 63: BMS2 Warning
   RUNG wire#powerrail
      { S7_Templates := "SrcType := Word" } NE_Contact(in1 := #BBwWarn1, in2 := 0)
      Coil( "BMS2".BBxWarnSt )
   END_RUNG
   // the same network as SCL:
   "BMS2".BBxWarnSt := #BBwWarn1 <> 0;
END_REGION

REGION Network 64 (SCL): Computing number of Rack in Fault
   "BMS2".iNRackFault := BOOL_TO_INT("BMS2".BR01xFltSt) +
                         BOOL_TO_INT("BMS2".BR02xFltSt) +
                         BOOL_TO_INT("BMS2".BR03xFltSt) +
                         BOOL_TO_INT("BMS2".BR04xFltSt) +
                         BOOL_TO_INT("BMS2".BR05xFltSt) +
                         BOOL_TO_INT("BMS2".BR06xFltSt) +
                         BOOL_TO_INT("BMS2".BR07xFltSt) +
                         BOOL_TO_INT("BMS2".BR08xFltSt) +
                         BOOL_TO_INT("BMS2".BR09xFltSt) +
                         BOOL_TO_INT("BMS2".BR10xFltSt);
END_REGION

REGION Network 65: BMS2 BR01 Fault SubSystem
   RUNG wire#powerrail
      Contact( #BR01wAlm2.%X2 )
      Contact( #BR01wAlm2.%X3 )
      wire#w1
      Coil( "BMS2".BR01xSSFltSt )
   END_RUNG
   RUNG wire#powerrail
      Contact( #BR01wAlm3.%X6 )
   END_RUNG wire#w1
   // the same network as SCL:
   "BMS2".BR01xSSFltSt := (#BR01wAlm2.%X2 AND #BR01wAlm2.%X3) OR #BR01wAlm3.%X6;
END_REGION

REGION Network 66: BMS2 BR01 Fault
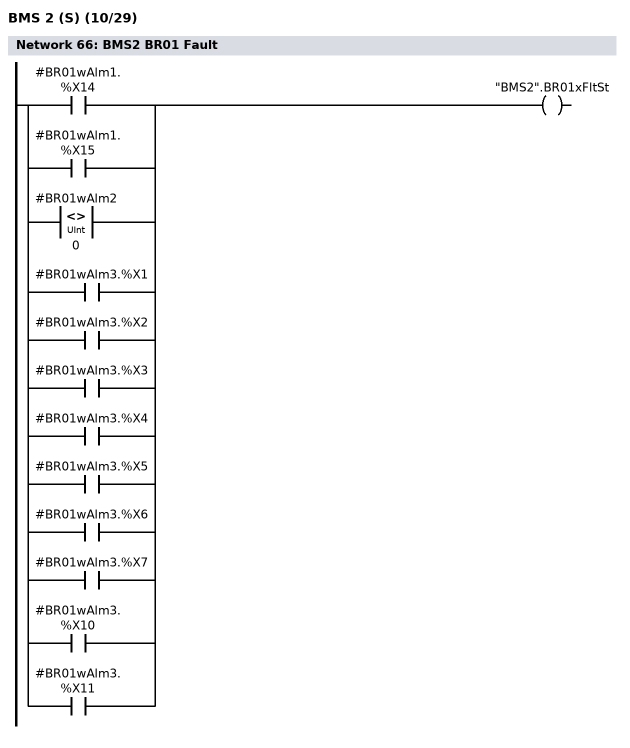
   RUNG wire#powerrail
      Contact( #BR01wAlm1.%X14 )
      wire#w1
      Coil( "BMS2".BR01xFltSt )
   END_RUNG
   RUNG wire#powerrail
      Contact( #BR01wAlm1.%X15 )
   END_RUNG wire#w1
   RUNG wire#powerrail
      { S7_Templates := "SrcType := UInt" } NE_Contact(in1 := #BR01wAlm2, in2 := 0)
   END_RUNG wire#w1
   RUNG wire#powerrail
      Contact( #BR01wAlm3.%X1 )
   END_RUNG wire#w1
   RUNG wire#powerrail
      Contact( #BR01wAlm3.%X2 )
   END_RUNG wire#w1
   RUNG wire#powerrail
      Contact( #BR01wAlm3.%X3 )
   END_RUNG wire#w1
   RUNG wire#powerrail
      Contact( #BR01wAlm3.%X4 )
   END_RUNG wire#w1
   RUNG wire#powerrail
      Contact( #BR01wAlm3.%X5 )
   END_RUNG wire#w1
   RUNG wire#powerrail
      Contact( #BR01wAlm3.%X6 )
   END_RUNG wire#w1
   RUNG wire#powerrail
      Contact( #BR01wAlm3.%X7 )
   END_RUNG wire#w1
   RUNG wire#powerrail
      Contact( #BR01wAlm3.%X10 )
   END_RUNG wire#w1
   RUNG wire#powerrail
      Contact( #BR01wAlm3.%X11 )
   END_RUNG wire#w1
   // the same network as SCL:
   "BMS2".BR01xFltSt := #BR01wAlm1.%X14 OR #BR01wAlm1.%X15 OR (#BR01wAlm2 <> 0) OR #BR01wAlm3.%X1 OR #BR01wAlm3.%X2 OR #BR01wAlm3.%X3 OR #BR01wAlm3.%X4 OR #BR01wAlm3.%X5 OR #BR01wAlm3.%X6 OR #BR01wAlm3.%X7 OR #BR01wAlm3.%X10 OR #BR01wAlm3.%X11;
END_REGION

REGION Network 67: BMS2 BR01 Alarm
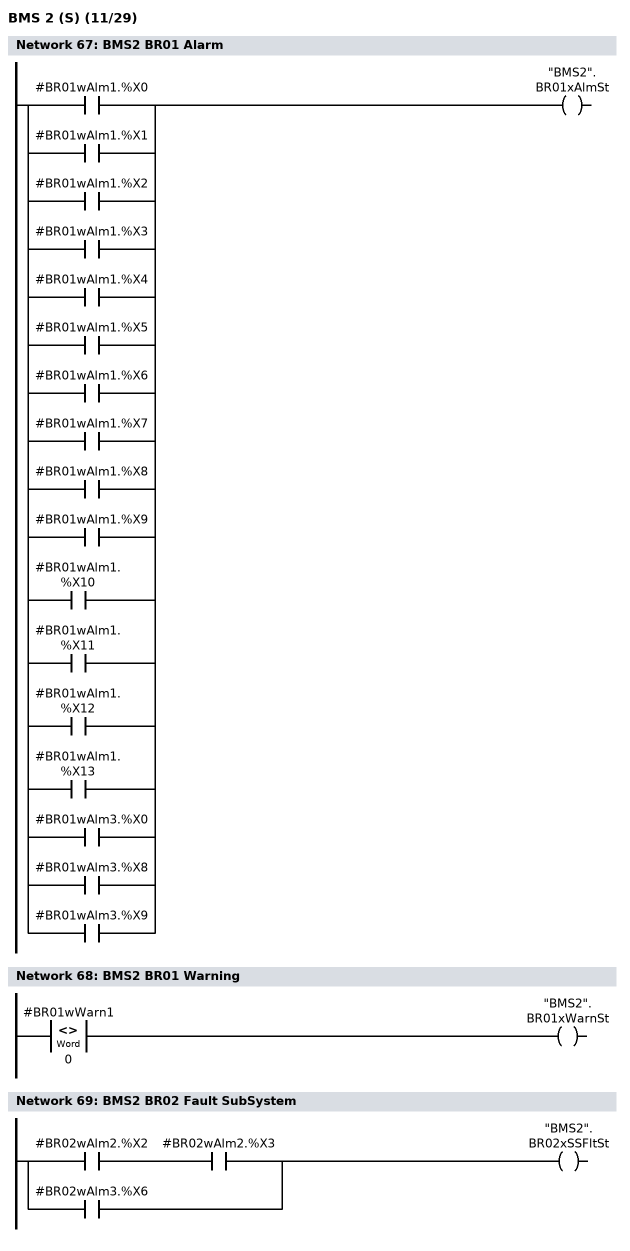
   RUNG wire#powerrail
      Contact( #BR01wAlm1.%X0 )
      wire#w1
      Coil( "BMS2".BR01xAlmSt )
   END_RUNG
   RUNG wire#powerrail
      Contact( #BR01wAlm1.%X1 )
   END_RUNG wire#w1
   RUNG wire#powerrail
      Contact( #BR01wAlm1.%X2 )
   END_RUNG wire#w1
   RUNG wire#powerrail
      Contact( #BR01wAlm1.%X3 )
   END_RUNG wire#w1
   RUNG wire#powerrail
      Contact( #BR01wAlm1.%X4 )
   END_RUNG wire#w1
   RUNG wire#powerrail
      Contact( #BR01wAlm1.%X5 )
   END_RUNG wire#w1
   RUNG wire#powerrail
      Contact( #BR01wAlm1.%X6 )
   END_RUNG wire#w1
   RUNG wire#powerrail
      Contact( #BR01wAlm1.%X7 )
   END_RUNG wire#w1
   RUNG wire#powerrail
      Contact( #BR01wAlm1.%X8 )
   END_RUNG wire#w1
   RUNG wire#powerrail
      Contact( #BR01wAlm1.%X9 )
   END_RUNG wire#w1
   RUNG wire#powerrail
      Contact( #BR01wAlm1.%X10 )
   END_RUNG wire#w1
   RUNG wire#powerrail
      Contact( #BR01wAlm1.%X11 )
   END_RUNG wire#w1
   RUNG wire#powerrail
      Contact( #BR01wAlm1.%X12 )
   END_RUNG wire#w1
   RUNG wire#powerrail
      Contact( #BR01wAlm1.%X13 )
   END_RUNG wire#w1
   RUNG wire#powerrail
      Contact( #BR01wAlm3.%X0 )
   END_RUNG wire#w1
   RUNG wire#powerrail
      Contact( #BR01wAlm3.%X8 )
   END_RUNG wire#w1
   RUNG wire#powerrail
      Contact( #BR01wAlm3.%X9 )
   END_RUNG wire#w1
   // the same network as SCL:
   "BMS2".BR01xAlmSt := #BR01wAlm1.%X0 OR #BR01wAlm1.%X1 OR #BR01wAlm1.%X2 OR #BR01wAlm1.%X3 OR #BR01wAlm1.%X4 OR #BR01wAlm1.%X5 OR #BR01wAlm1.%X6 OR #BR01wAlm1.%X7 OR #BR01wAlm1.%X8 OR #BR01wAlm1.%X9 OR #BR01wAlm1.%X10 OR #BR01wAlm1.%X11 OR #BR01wAlm1.%X12 OR #BR01wAlm1.%X13 OR #BR01wAlm3.%X0 OR #BR01wAlm3.%X8 OR #BR01wAlm3.%X9;
END_REGION

REGION Network 68: BMS2 BR01 Warning
   RUNG wire#powerrail
      { S7_Templates := "SrcType := Word" } NE_Contact(in1 := #BR01wWarn1, in2 := 0)
      Coil( "BMS2".BR01xWarnSt )
   END_RUNG
   // the same network as SCL:
   "BMS2".BR01xWarnSt := #BR01wWarn1 <> 0;
END_REGION

REGION Network 69: BMS2 BR02 Fault SubSystem
   RUNG wire#powerrail
      Contact( #BR02wAlm2.%X2 )
      Contact( #BR02wAlm2.%X3 )
      wire#w1
      Coil( "BMS2".BR02xSSFltSt )
   END_RUNG
   RUNG wire#powerrail
      Contact( #BR02wAlm3.%X6 )
   END_RUNG wire#w1
   // the same network as SCL:
   "BMS2".BR02xSSFltSt := (#BR02wAlm2.%X2 AND #BR02wAlm2.%X3) OR #BR02wAlm3.%X6;
END_REGION

REGION Network 70: BMS2 BR02 Fault
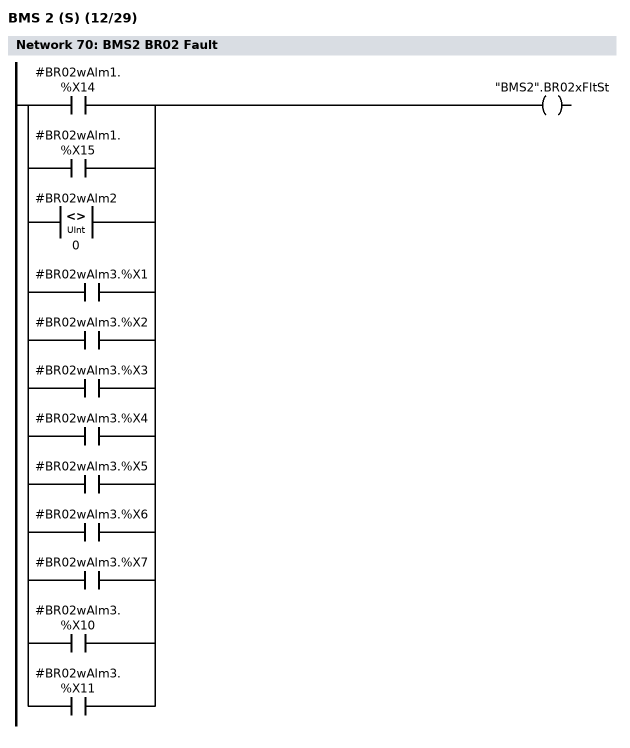
   RUNG wire#powerrail
      Contact( #BR02wAlm1.%X14 )
      wire#w1
      Coil( "BMS2".BR02xFltSt )
   END_RUNG
   RUNG wire#powerrail
      Contact( #BR02wAlm1.%X15 )
   END_RUNG wire#w1
   RUNG wire#powerrail
      { S7_Templates := "SrcType := UInt" } NE_Contact(in1 := #BR02wAlm2, in2 := 0)
   END_RUNG wire#w1
   RUNG wire#powerrail
      Contact( #BR02wAlm3.%X1 )
   END_RUNG wire#w1
   RUNG wire#powerrail
      Contact( #BR02wAlm3.%X2 )
   END_RUNG wire#w1
   RUNG wire#powerrail
      Contact( #BR02wAlm3.%X3 )
   END_RUNG wire#w1
   RUNG wire#powerrail
      Contact( #BR02wAlm3.%X4 )
   END_RUNG wire#w1
   RUNG wire#powerrail
      Contact( #BR02wAlm3.%X5 )
   END_RUNG wire#w1
   RUNG wire#powerrail
      Contact( #BR02wAlm3.%X6 )
   END_RUNG wire#w1
   RUNG wire#powerrail
      Contact( #BR02wAlm3.%X7 )
   END_RUNG wire#w1
   RUNG wire#powerrail
      Contact( #BR02wAlm3.%X10 )
   END_RUNG wire#w1
   RUNG wire#powerrail
      Contact( #BR02wAlm3.%X11 )
   END_RUNG wire#w1
   // the same network as SCL:
   "BMS2".BR02xFltSt := #BR02wAlm1.%X14 OR #BR02wAlm1.%X15 OR (#BR02wAlm2 <> 0) OR #BR02wAlm3.%X1 OR #BR02wAlm3.%X2 OR #BR02wAlm3.%X3 OR #BR02wAlm3.%X4 OR #BR02wAlm3.%X5 OR #BR02wAlm3.%X6 OR #BR02wAlm3.%X7 OR #BR02wAlm3.%X10 OR #BR02wAlm3.%X11;
END_REGION

REGION Network 71: BMS2 BR02 Alarm
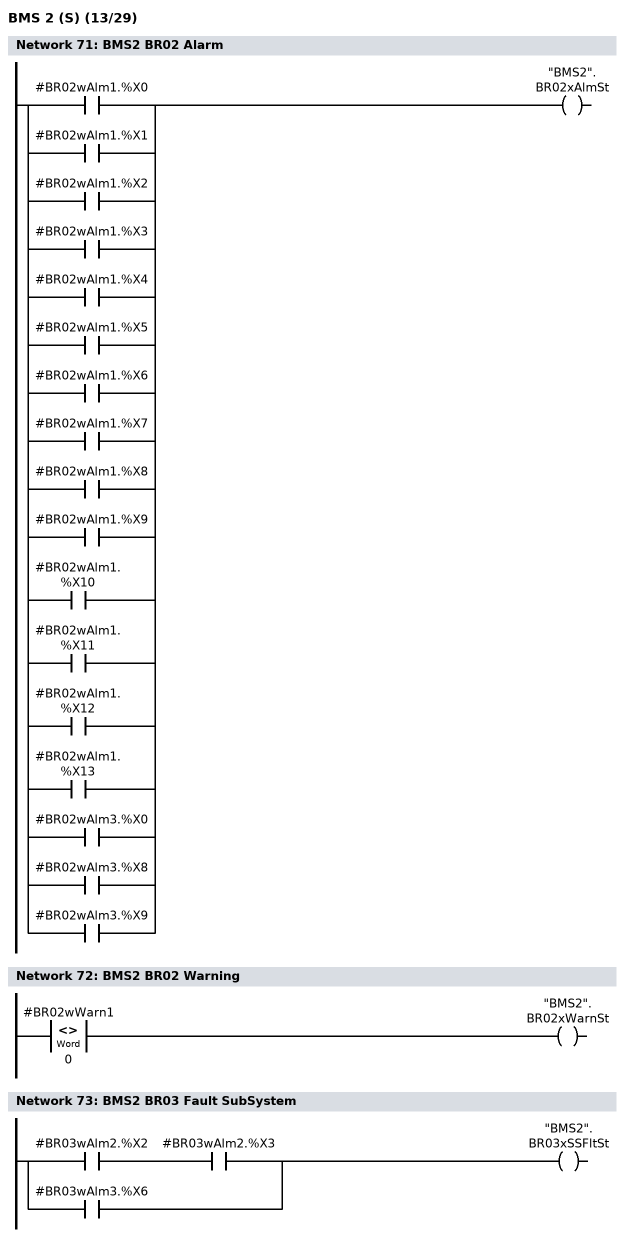
   RUNG wire#powerrail
      Contact( #BR02wAlm1.%X0 )
      wire#w1
      Coil( "BMS2".BR02xAlmSt )
   END_RUNG
   RUNG wire#powerrail
      Contact( #BR02wAlm1.%X1 )
   END_RUNG wire#w1
   RUNG wire#powerrail
      Contact( #BR02wAlm1.%X2 )
   END_RUNG wire#w1
   RUNG wire#powerrail
      Contact( #BR02wAlm1.%X3 )
   END_RUNG wire#w1
   RUNG wire#powerrail
      Contact( #BR02wAlm1.%X4 )
   END_RUNG wire#w1
   RUNG wire#powerrail
      Contact( #BR02wAlm1.%X5 )
   END_RUNG wire#w1
   RUNG wire#powerrail
      Contact( #BR02wAlm1.%X6 )
   END_RUNG wire#w1
   RUNG wire#powerrail
      Contact( #BR02wAlm1.%X7 )
   END_RUNG wire#w1
   RUNG wire#powerrail
      Contact( #BR02wAlm1.%X8 )
   END_RUNG wire#w1
   RUNG wire#powerrail
      Contact( #BR02wAlm1.%X9 )
   END_RUNG wire#w1
   RUNG wire#powerrail
      Contact( #BR02wAlm1.%X10 )
   END_RUNG wire#w1
   RUNG wire#powerrail
      Contact( #BR02wAlm1.%X11 )
   END_RUNG wire#w1
   RUNG wire#powerrail
      Contact( #BR02wAlm1.%X12 )
   END_RUNG wire#w1
   RUNG wire#powerrail
      Contact( #BR02wAlm1.%X13 )
   END_RUNG wire#w1
   RUNG wire#powerrail
      Contact( #BR02wAlm3.%X0 )
   END_RUNG wire#w1
   RUNG wire#powerrail
      Contact( #BR02wAlm3.%X8 )
   END_RUNG wire#w1
   RUNG wire#powerrail
      Contact( #BR02wAlm3.%X9 )
   END_RUNG wire#w1
   // the same network as SCL:
   "BMS2".BR02xAlmSt := #BR02wAlm1.%X0 OR #BR02wAlm1.%X1 OR #BR02wAlm1.%X2 OR #BR02wAlm1.%X3 OR #BR02wAlm1.%X4 OR #BR02wAlm1.%X5 OR #BR02wAlm1.%X6 OR #BR02wAlm1.%X7 OR #BR02wAlm1.%X8 OR #BR02wAlm1.%X9 OR #BR02wAlm1.%X10 OR #BR02wAlm1.%X11 OR #BR02wAlm1.%X12 OR #BR02wAlm1.%X13 OR #BR02wAlm3.%X0 OR #BR02wAlm3.%X8 OR #BR02wAlm3.%X9;
END_REGION

REGION Network 72: BMS2 BR02 Warning
   RUNG wire#powerrail
      { S7_Templates := "SrcType := Word" } NE_Contact(in1 := #BR02wWarn1, in2 := 0)
      Coil( "BMS2".BR02xWarnSt )
   END_RUNG
   // the same network as SCL:
   "BMS2".BR02xWarnSt := #BR02wWarn1 <> 0;
END_REGION

REGION Network 73: BMS2 BR03 Fault SubSystem
   RUNG wire#powerrail
      Contact( #BR03wAlm2.%X2 )
      Contact( #BR03wAlm2.%X3 )
      wire#w1
      Coil( "BMS2".BR03xSSFltSt )
   END_RUNG
   RUNG wire#powerrail
      Contact( #BR03wAlm3.%X6 )
   END_RUNG wire#w1
   // the same network as SCL:
   "BMS2".BR03xSSFltSt := (#BR03wAlm2.%X2 AND #BR03wAlm2.%X3) OR #BR03wAlm3.%X6;
END_REGION

REGION Network 74: BMS2 BR03 Fault
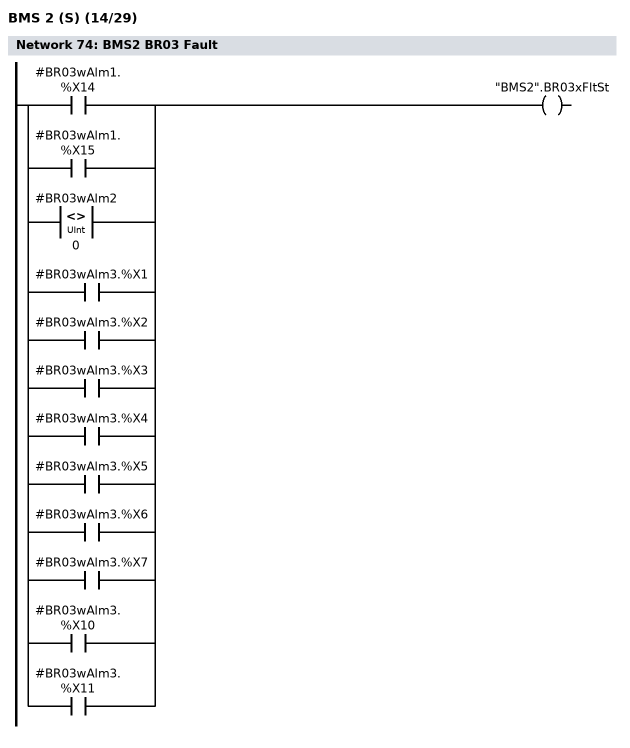
   RUNG wire#powerrail
      Contact( #BR03wAlm1.%X14 )
      wire#w1
      Coil( "BMS2".BR03xFltSt )
   END_RUNG
   RUNG wire#powerrail
      Contact( #BR03wAlm1.%X15 )
   END_RUNG wire#w1
   RUNG wire#powerrail
      { S7_Templates := "SrcType := UInt" } NE_Contact(in1 := #BR03wAlm2, in2 := 0)
   END_RUNG wire#w1
   RUNG wire#powerrail
      Contact( #BR03wAlm3.%X1 )
   END_RUNG wire#w1
   RUNG wire#powerrail
      Contact( #BR03wAlm3.%X2 )
   END_RUNG wire#w1
   RUNG wire#powerrail
      Contact( #BR03wAlm3.%X3 )
   END_RUNG wire#w1
   RUNG wire#powerrail
      Contact( #BR03wAlm3.%X4 )
   END_RUNG wire#w1
   RUNG wire#powerrail
      Contact( #BR03wAlm3.%X5 )
   END_RUNG wire#w1
   RUNG wire#powerrail
      Contact( #BR03wAlm3.%X6 )
   END_RUNG wire#w1
   RUNG wire#powerrail
      Contact( #BR03wAlm3.%X7 )
   END_RUNG wire#w1
   RUNG wire#powerrail
      Contact( #BR03wAlm3.%X10 )
   END_RUNG wire#w1
   RUNG wire#powerrail
      Contact( #BR03wAlm3.%X11 )
   END_RUNG wire#w1
   // the same network as SCL:
   "BMS2".BR03xFltSt := #BR03wAlm1.%X14 OR #BR03wAlm1.%X15 OR (#BR03wAlm2 <> 0) OR #BR03wAlm3.%X1 OR #BR03wAlm3.%X2 OR #BR03wAlm3.%X3 OR #BR03wAlm3.%X4 OR #BR03wAlm3.%X5 OR #BR03wAlm3.%X6 OR #BR03wAlm3.%X7 OR #BR03wAlm3.%X10 OR #BR03wAlm3.%X11;
END_REGION

REGION Network 75: BMS2 BR03 Alarm
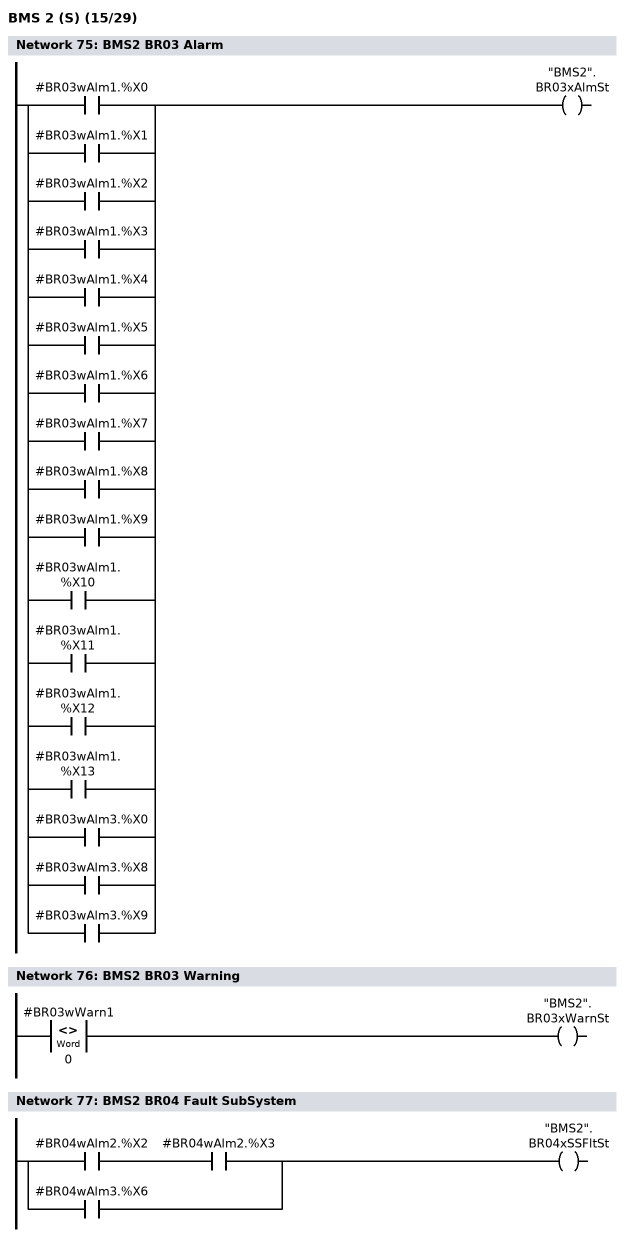
   RUNG wire#powerrail
      Contact( #BR03wAlm1.%X0 )
      wire#w1
      Coil( "BMS2".BR03xAlmSt )
   END_RUNG
   RUNG wire#powerrail
      Contact( #BR03wAlm1.%X1 )
   END_RUNG wire#w1
   RUNG wire#powerrail
      Contact( #BR03wAlm1.%X2 )
   END_RUNG wire#w1
   RUNG wire#powerrail
      Contact( #BR03wAlm1.%X3 )
   END_RUNG wire#w1
   RUNG wire#powerrail
      Contact( #BR03wAlm1.%X4 )
   END_RUNG wire#w1
   RUNG wire#powerrail
      Contact( #BR03wAlm1.%X5 )
   END_RUNG wire#w1
   RUNG wire#powerrail
      Contact( #BR03wAlm1.%X6 )
   END_RUNG wire#w1
   RUNG wire#powerrail
      Contact( #BR03wAlm1.%X7 )
   END_RUNG wire#w1
   RUNG wire#powerrail
      Contact( #BR03wAlm1.%X8 )
   END_RUNG wire#w1
   RUNG wire#powerrail
      Contact( #BR03wAlm1.%X9 )
   END_RUNG wire#w1
   RUNG wire#powerrail
      Contact( #BR03wAlm1.%X10 )
   END_RUNG wire#w1
   RUNG wire#powerrail
      Contact( #BR03wAlm1.%X11 )
   END_RUNG wire#w1
   RUNG wire#powerrail
      Contact( #BR03wAlm1.%X12 )
   END_RUNG wire#w1
   RUNG wire#powerrail
      Contact( #BR03wAlm1.%X13 )
   END_RUNG wire#w1
   RUNG wire#powerrail
      Contact( #BR03wAlm3.%X0 )
   END_RUNG wire#w1
   RUNG wire#powerrail
      Contact( #BR03wAlm3.%X8 )
   END_RUNG wire#w1
   RUNG wire#powerrail
      Contact( #BR03wAlm3.%X9 )
   END_RUNG wire#w1
   // the same network as SCL:
   "BMS2".BR03xAlmSt := #BR03wAlm1.%X0 OR #BR03wAlm1.%X1 OR #BR03wAlm1.%X2 OR #BR03wAlm1.%X3 OR #BR03wAlm1.%X4 OR #BR03wAlm1.%X5 OR #BR03wAlm1.%X6 OR #BR03wAlm1.%X7 OR #BR03wAlm1.%X8 OR #BR03wAlm1.%X9 OR #BR03wAlm1.%X10 OR #BR03wAlm1.%X11 OR #BR03wAlm1.%X12 OR #BR03wAlm1.%X13 OR #BR03wAlm3.%X0 OR #BR03wAlm3.%X8 OR #BR03wAlm3.%X9;
END_REGION

REGION Network 76: BMS2 BR03 Warning
   RUNG wire#powerrail
      { S7_Templates := "SrcType := Word" } NE_Contact(in1 := #BR03wWarn1, in2 := 0)
      Coil( "BMS2".BR03xWarnSt )
   END_RUNG
   // the same network as SCL:
   "BMS2".BR03xWarnSt := #BR03wWarn1 <> 0;
END_REGION

REGION Network 77: BMS2 BR04 Fault SubSystem
   RUNG wire#powerrail
      Contact( #BR04wAlm2.%X2 )
      Contact( #BR04wAlm2.%X3 )
      wire#w1
      Coil( "BMS2".BR04xSSFltSt )
   END_RUNG
   RUNG wire#powerrail
      Contact( #BR04wAlm3.%X6 )
   END_RUNG wire#w1
   // the same network as SCL:
   "BMS2".BR04xSSFltSt := (#BR04wAlm2.%X2 AND #BR04wAlm2.%X3) OR #BR04wAlm3.%X6;
END_REGION

REGION Network 78: BMS2 BR04 Fault
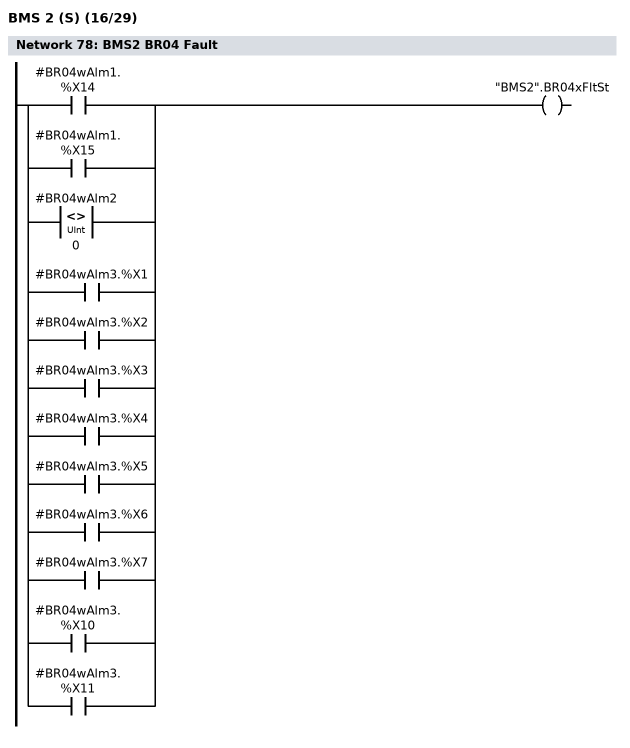
   RUNG wire#powerrail
      Contact( #BR04wAlm1.%X14 )
      wire#w1
      Coil( "BMS2".BR04xFltSt )
   END_RUNG
   RUNG wire#powerrail
      Contact( #BR04wAlm1.%X15 )
   END_RUNG wire#w1
   RUNG wire#powerrail
      { S7_Templates := "SrcType := UInt" } NE_Contact(in1 := #BR04wAlm2, in2 := 0)
   END_RUNG wire#w1
   RUNG wire#powerrail
      Contact( #BR04wAlm3.%X1 )
   END_RUNG wire#w1
   RUNG wire#powerrail
      Contact( #BR04wAlm3.%X2 )
   END_RUNG wire#w1
   RUNG wire#powerrail
      Contact( #BR04wAlm3.%X3 )
   END_RUNG wire#w1
   RUNG wire#powerrail
      Contact( #BR04wAlm3.%X4 )
   END_RUNG wire#w1
   RUNG wire#powerrail
      Contact( #BR04wAlm3.%X5 )
   END_RUNG wire#w1
   RUNG wire#powerrail
      Contact( #BR04wAlm3.%X6 )
   END_RUNG wire#w1
   RUNG wire#powerrail
      Contact( #BR04wAlm3.%X7 )
   END_RUNG wire#w1
   RUNG wire#powerrail
      Contact( #BR04wAlm3.%X10 )
   END_RUNG wire#w1
   RUNG wire#powerrail
      Contact( #BR04wAlm3.%X11 )
   END_RUNG wire#w1
   // the same network as SCL:
   "BMS2".BR04xFltSt := #BR04wAlm1.%X14 OR #BR04wAlm1.%X15 OR (#BR04wAlm2 <> 0) OR #BR04wAlm3.%X1 OR #BR04wAlm3.%X2 OR #BR04wAlm3.%X3 OR #BR04wAlm3.%X4 OR #BR04wAlm3.%X5 OR #BR04wAlm3.%X6 OR #BR04wAlm3.%X7 OR #BR04wAlm3.%X10 OR #BR04wAlm3.%X11;
END_REGION

REGION Network 79: BMS2 BR04 Alarm
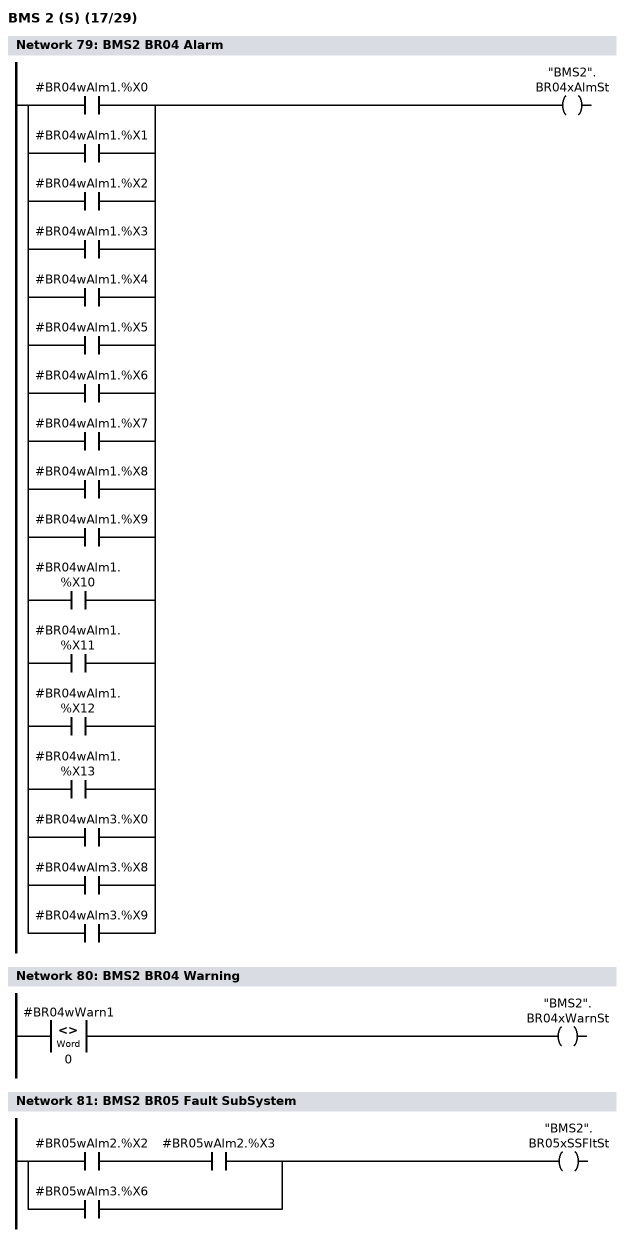
   RUNG wire#powerrail
      Contact( #BR04wAlm1.%X0 )
      wire#w1
      Coil( "BMS2".BR04xAlmSt )
   END_RUNG
   RUNG wire#powerrail
      Contact( #BR04wAlm1.%X1 )
   END_RUNG wire#w1
   RUNG wire#powerrail
      Contact( #BR04wAlm1.%X2 )
   END_RUNG wire#w1
   RUNG wire#powerrail
      Contact( #BR04wAlm1.%X3 )
   END_RUNG wire#w1
   RUNG wire#powerrail
      Contact( #BR04wAlm1.%X4 )
   END_RUNG wire#w1
   RUNG wire#powerrail
      Contact( #BR04wAlm1.%X5 )
   END_RUNG wire#w1
   RUNG wire#powerrail
      Contact( #BR04wAlm1.%X6 )
   END_RUNG wire#w1
   RUNG wire#powerrail
      Contact( #BR04wAlm1.%X7 )
   END_RUNG wire#w1
   RUNG wire#powerrail
      Contact( #BR04wAlm1.%X8 )
   END_RUNG wire#w1
   RUNG wire#powerrail
      Contact( #BR04wAlm1.%X9 )
   END_RUNG wire#w1
   RUNG wire#powerrail
      Contact( #BR04wAlm1.%X10 )
   END_RUNG wire#w1
   RUNG wire#powerrail
      Contact( #BR04wAlm1.%X11 )
   END_RUNG wire#w1
   RUNG wire#powerrail
      Contact( #BR04wAlm1.%X12 )
   END_RUNG wire#w1
   RUNG wire#powerrail
      Contact( #BR04wAlm1.%X13 )
   END_RUNG wire#w1
   RUNG wire#powerrail
      Contact( #BR04wAlm3.%X0 )
   END_RUNG wire#w1
   RUNG wire#powerrail
      Contact( #BR04wAlm3.%X8 )
   END_RUNG wire#w1
   RUNG wire#powerrail
      Contact( #BR04wAlm3.%X9 )
   END_RUNG wire#w1
   // the same network as SCL:
   "BMS2".BR04xAlmSt := #BR04wAlm1.%X0 OR #BR04wAlm1.%X1 OR #BR04wAlm1.%X2 OR #BR04wAlm1.%X3 OR #BR04wAlm1.%X4 OR #BR04wAlm1.%X5 OR #BR04wAlm1.%X6 OR #BR04wAlm1.%X7 OR #BR04wAlm1.%X8 OR #BR04wAlm1.%X9 OR #BR04wAlm1.%X10 OR #BR04wAlm1.%X11 OR #BR04wAlm1.%X12 OR #BR04wAlm1.%X13 OR #BR04wAlm3.%X0 OR #BR04wAlm3.%X8 OR #BR04wAlm3.%X9;
END_REGION

REGION Network 80: BMS2 BR04 Warning
   RUNG wire#powerrail
      { S7_Templates := "SrcType := Word" } NE_Contact(in1 := #BR04wWarn1, in2 := 0)
      Coil( "BMS2".BR04xWarnSt )
   END_RUNG
   // the same network as SCL:
   "BMS2".BR04xWarnSt := #BR04wWarn1 <> 0;
END_REGION

REGION Network 81: BMS2 BR05 Fault SubSystem
   RUNG wire#powerrail
      Contact( #BR05wAlm2.%X2 )
      Contact( #BR05wAlm2.%X3 )
      wire#w1
      Coil( "BMS2".BR05xSSFltSt )
   END_RUNG
   RUNG wire#powerrail
      Contact( #BR05wAlm3.%X6 )
   END_RUNG wire#w1
   // the same network as SCL:
   "BMS2".BR05xSSFltSt := (#BR05wAlm2.%X2 AND #BR05wAlm2.%X3) OR #BR05wAlm3.%X6;
END_REGION

REGION Network 82: BMS2 BR05 Fault
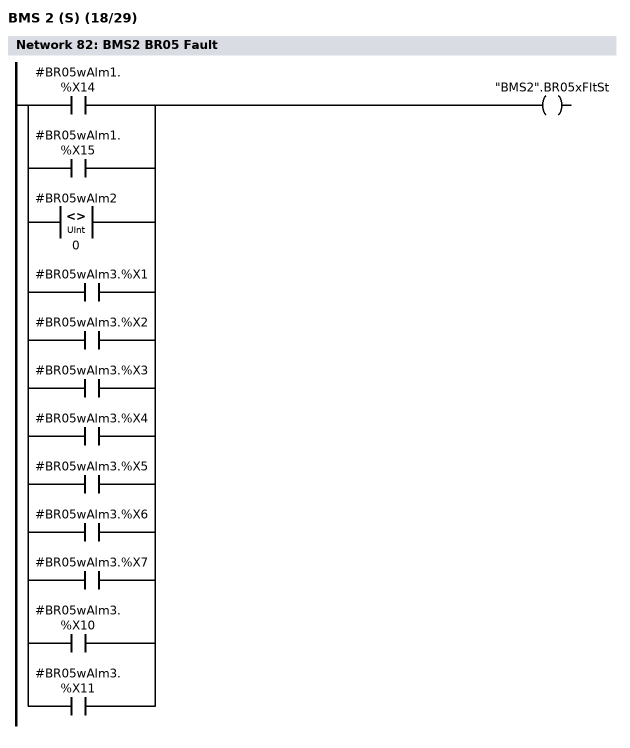
   RUNG wire#powerrail
      Contact( #BR05wAlm1.%X14 )
      wire#w1
      Coil( "BMS2".BR05xFltSt )
   END_RUNG
   RUNG wire#powerrail
      Contact( #BR05wAlm1.%X15 )
   END_RUNG wire#w1
   RUNG wire#powerrail
      { S7_Templates := "SrcType := UInt" } NE_Contact(in1 := #BR05wAlm2, in2 := 0)
   END_RUNG wire#w1
   RUNG wire#powerrail
      Contact( #BR05wAlm3.%X1 )
   END_RUNG wire#w1
   RUNG wire#powerrail
      Contact( #BR05wAlm3.%X2 )
   END_RUNG wire#w1
   RUNG wire#powerrail
      Contact( #BR05wAlm3.%X3 )
   END_RUNG wire#w1
   RUNG wire#powerrail
      Contact( #BR05wAlm3.%X4 )
   END_RUNG wire#w1
   RUNG wire#powerrail
      Contact( #BR05wAlm3.%X5 )
   END_RUNG wire#w1
   RUNG wire#powerrail
      Contact( #BR05wAlm3.%X6 )
   END_RUNG wire#w1
   RUNG wire#powerrail
      Contact( #BR05wAlm3.%X7 )
   END_RUNG wire#w1
   RUNG wire#powerrail
      Contact( #BR05wAlm3.%X10 )
   END_RUNG wire#w1
   RUNG wire#powerrail
      Contact( #BR05wAlm3.%X11 )
   END_RUNG wire#w1
   // the same network as SCL:
   "BMS2".BR05xFltSt := #BR05wAlm1.%X14 OR #BR05wAlm1.%X15 OR (#BR05wAlm2 <> 0) OR #BR05wAlm3.%X1 OR #BR05wAlm3.%X2 OR #BR05wAlm3.%X3 OR #BR05wAlm3.%X4 OR #BR05wAlm3.%X5 OR #BR05wAlm3.%X6 OR #BR05wAlm3.%X7 OR #BR05wAlm3.%X10 OR #BR05wAlm3.%X11;
END_REGION

REGION Network 83: BMS2 BR05 Alarm
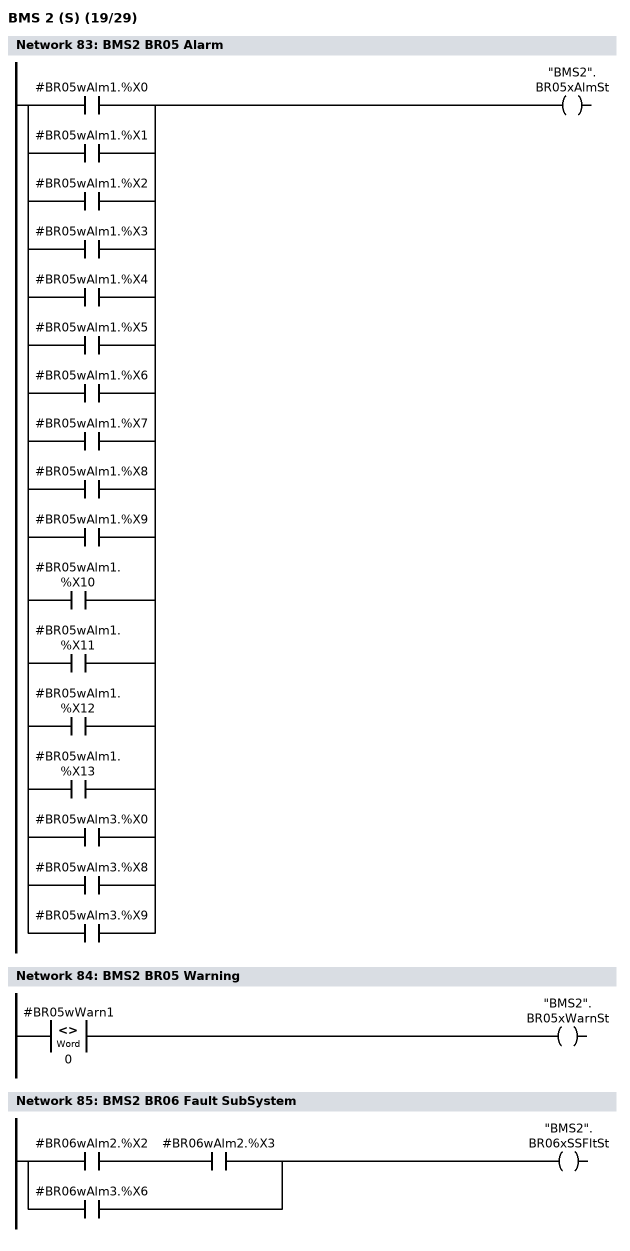
   RUNG wire#powerrail
      Contact( #BR05wAlm1.%X0 )
      wire#w1
      Coil( "BMS2".BR05xAlmSt )
   END_RUNG
   RUNG wire#powerrail
      Contact( #BR05wAlm1.%X1 )
   END_RUNG wire#w1
   RUNG wire#powerrail
      Contact( #BR05wAlm1.%X2 )
   END_RUNG wire#w1
   RUNG wire#powerrail
      Contact( #BR05wAlm1.%X3 )
   END_RUNG wire#w1
   RUNG wire#powerrail
      Contact( #BR05wAlm1.%X4 )
   END_RUNG wire#w1
   RUNG wire#powerrail
      Contact( #BR05wAlm1.%X5 )
   END_RUNG wire#w1
   RUNG wire#powerrail
      Contact( #BR05wAlm1.%X6 )
   END_RUNG wire#w1
   RUNG wire#powerrail
      Contact( #BR05wAlm1.%X7 )
   END_RUNG wire#w1
   RUNG wire#powerrail
      Contact( #BR05wAlm1.%X8 )
   END_RUNG wire#w1
   RUNG wire#powerrail
      Contact( #BR05wAlm1.%X9 )
   END_RUNG wire#w1
   RUNG wire#powerrail
      Contact( #BR05wAlm1.%X10 )
   END_RUNG wire#w1
   RUNG wire#powerrail
      Contact( #BR05wAlm1.%X11 )
   END_RUNG wire#w1
   RUNG wire#powerrail
      Contact( #BR05wAlm1.%X12 )
   END_RUNG wire#w1
   RUNG wire#powerrail
      Contact( #BR05wAlm1.%X13 )
   END_RUNG wire#w1
   RUNG wire#powerrail
      Contact( #BR05wAlm3.%X0 )
   END_RUNG wire#w1
   RUNG wire#powerrail
      Contact( #BR05wAlm3.%X8 )
   END_RUNG wire#w1
   RUNG wire#powerrail
      Contact( #BR05wAlm3.%X9 )
   END_RUNG wire#w1
   // the same network as SCL:
   "BMS2".BR05xAlmSt := #BR05wAlm1.%X0 OR #BR05wAlm1.%X1 OR #BR05wAlm1.%X2 OR #BR05wAlm1.%X3 OR #BR05wAlm1.%X4 OR #BR05wAlm1.%X5 OR #BR05wAlm1.%X6 OR #BR05wAlm1.%X7 OR #BR05wAlm1.%X8 OR #BR05wAlm1.%X9 OR #BR05wAlm1.%X10 OR #BR05wAlm1.%X11 OR #BR05wAlm1.%X12 OR #BR05wAlm1.%X13 OR #BR05wAlm3.%X0 OR #BR05wAlm3.%X8 OR #BR05wAlm3.%X9;
END_REGION

REGION Network 84: BMS2 BR05 Warning
   RUNG wire#powerrail
      { S7_Templates := "SrcType := Word" } NE_Contact(in1 := #BR05wWarn1, in2 := 0)
      Coil( "BMS2".BR05xWarnSt )
   END_RUNG
   // the same network as SCL:
   "BMS2".BR05xWarnSt := #BR05wWarn1 <> 0;
END_REGION

REGION Network 85: BMS2 BR06 Fault SubSystem
   RUNG wire#powerrail
      Contact( #BR06wAlm2.%X2 )
      Contact( #BR06wAlm2.%X3 )
      wire#w1
      Coil( "BMS2".BR06xSSFltSt )
   END_RUNG
   RUNG wire#powerrail
      Contact( #BR06wAlm3.%X6 )
   END_RUNG wire#w1
   // the same network as SCL:
   "BMS2".BR06xSSFltSt := (#BR06wAlm2.%X2 AND #BR06wAlm2.%X3) OR #BR06wAlm3.%X6;
END_REGION

REGION Network 86: BMS2 BR06 Fault
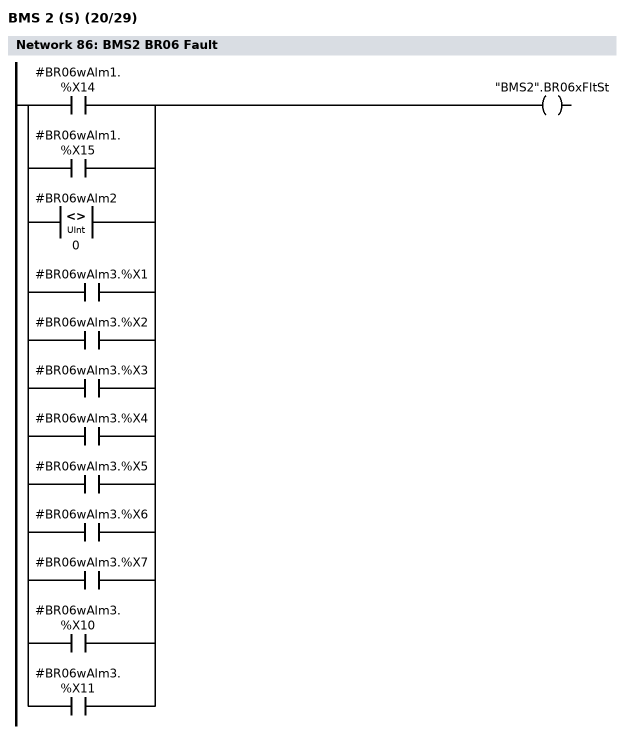
   RUNG wire#powerrail
      Contact( #BR06wAlm1.%X14 )
      wire#w1
      Coil( "BMS2".BR06xFltSt )
   END_RUNG
   RUNG wire#powerrail
      Contact( #BR06wAlm1.%X15 )
   END_RUNG wire#w1
   RUNG wire#powerrail
      { S7_Templates := "SrcType := UInt" } NE_Contact(in1 := #BR06wAlm2, in2 := 0)
   END_RUNG wire#w1
   RUNG wire#powerrail
      Contact( #BR06wAlm3.%X1 )
   END_RUNG wire#w1
   RUNG wire#powerrail
      Contact( #BR06wAlm3.%X2 )
   END_RUNG wire#w1
   RUNG wire#powerrail
      Contact( #BR06wAlm3.%X3 )
   END_RUNG wire#w1
   RUNG wire#powerrail
      Contact( #BR06wAlm3.%X4 )
   END_RUNG wire#w1
   RUNG wire#powerrail
      Contact( #BR06wAlm3.%X5 )
   END_RUNG wire#w1
   RUNG wire#powerrail
      Contact( #BR06wAlm3.%X6 )
   END_RUNG wire#w1
   RUNG wire#powerrail
      Contact( #BR06wAlm3.%X7 )
   END_RUNG wire#w1
   RUNG wire#powerrail
      Contact( #BR06wAlm3.%X10 )
   END_RUNG wire#w1
   RUNG wire#powerrail
      Contact( #BR06wAlm3.%X11 )
   END_RUNG wire#w1
   // the same network as SCL:
   "BMS2".BR06xFltSt := #BR06wAlm1.%X14 OR #BR06wAlm1.%X15 OR (#BR06wAlm2 <> 0) OR #BR06wAlm3.%X1 OR #BR06wAlm3.%X2 OR #BR06wAlm3.%X3 OR #BR06wAlm3.%X4 OR #BR06wAlm3.%X5 OR #BR06wAlm3.%X6 OR #BR06wAlm3.%X7 OR #BR06wAlm3.%X10 OR #BR06wAlm3.%X11;
END_REGION

REGION Network 87: BMS2 BR06 Alarm
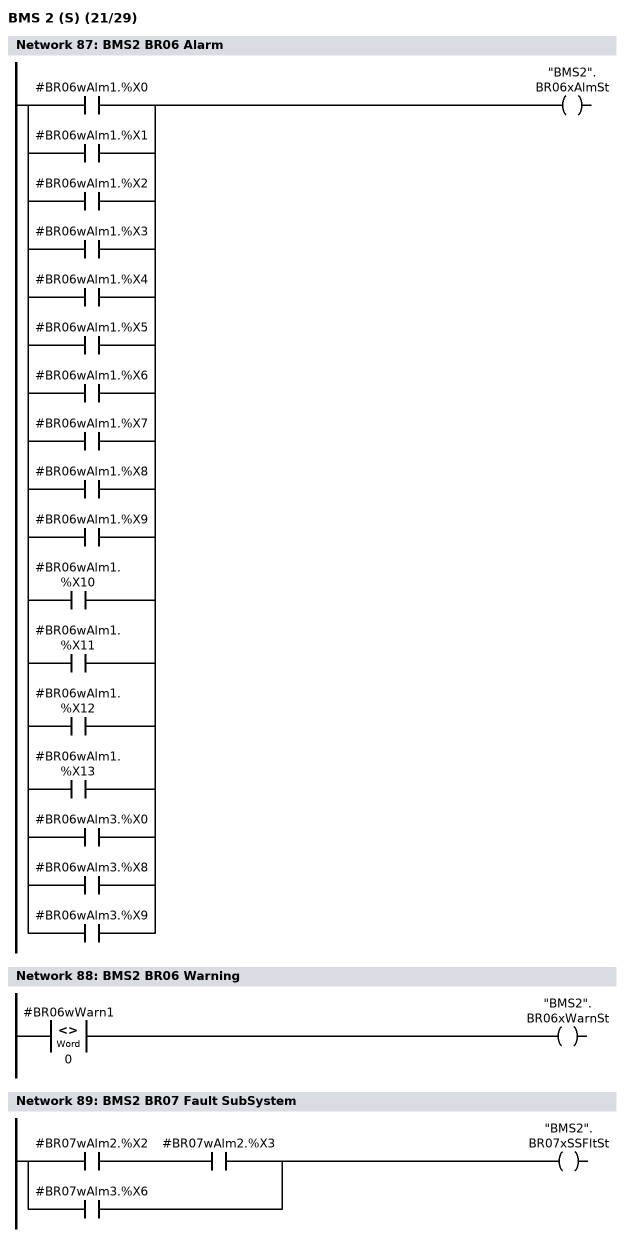
   RUNG wire#powerrail
      Contact( #BR06wAlm1.%X0 )
      wire#w1
      Coil( "BMS2".BR06xAlmSt )
   END_RUNG
   RUNG wire#powerrail
      Contact( #BR06wAlm1.%X1 )
   END_RUNG wire#w1
   RUNG wire#powerrail
      Contact( #BR06wAlm1.%X2 )
   END_RUNG wire#w1
   RUNG wire#powerrail
      Contact( #BR06wAlm1.%X3 )
   END_RUNG wire#w1
   RUNG wire#powerrail
      Contact( #BR06wAlm1.%X4 )
   END_RUNG wire#w1
   RUNG wire#powerrail
      Contact( #BR06wAlm1.%X5 )
   END_RUNG wire#w1
   RUNG wire#powerrail
      Contact( #BR06wAlm1.%X6 )
   END_RUNG wire#w1
   RUNG wire#powerrail
      Contact( #BR06wAlm1.%X7 )
   END_RUNG wire#w1
   RUNG wire#powerrail
      Contact( #BR06wAlm1.%X8 )
   END_RUNG wire#w1
   RUNG wire#powerrail
      Contact( #BR06wAlm1.%X9 )
   END_RUNG wire#w1
   RUNG wire#powerrail
      Contact( #BR06wAlm1.%X10 )
   END_RUNG wire#w1
   RUNG wire#powerrail
      Contact( #BR06wAlm1.%X11 )
   END_RUNG wire#w1
   RUNG wire#powerrail
      Contact( #BR06wAlm1.%X12 )
   END_RUNG wire#w1
   RUNG wire#powerrail
      Contact( #BR06wAlm1.%X13 )
   END_RUNG wire#w1
   RUNG wire#powerrail
      Contact( #BR06wAlm3.%X0 )
   END_RUNG wire#w1
   RUNG wire#powerrail
      Contact( #BR06wAlm3.%X8 )
   END_RUNG wire#w1
   RUNG wire#powerrail
      Contact( #BR06wAlm3.%X9 )
   END_RUNG wire#w1
   // the same network as SCL:
   "BMS2".BR06xAlmSt := #BR06wAlm1.%X0 OR #BR06wAlm1.%X1 OR #BR06wAlm1.%X2 OR #BR06wAlm1.%X3 OR #BR06wAlm1.%X4 OR #BR06wAlm1.%X5 OR #BR06wAlm1.%X6 OR #BR06wAlm1.%X7 OR #BR06wAlm1.%X8 OR #BR06wAlm1.%X9 OR #BR06wAlm1.%X10 OR #BR06wAlm1.%X11 OR #BR06wAlm1.%X12 OR #BR06wAlm1.%X13 OR #BR06wAlm3.%X0 OR #BR06wAlm3.%X8 OR #BR06wAlm3.%X9;
END_REGION

REGION Network 88: BMS2 BR06 Warning
   RUNG wire#powerrail
      { S7_Templates := "SrcType := Word" } NE_Contact(in1 := #BR06wWarn1, in2 := 0)
      Coil( "BMS2".BR06xWarnSt )
   END_RUNG
   // the same network as SCL:
   "BMS2".BR06xWarnSt := #BR06wWarn1 <> 0;
END_REGION

REGION Network 89: BMS2 BR07 Fault SubSystem
   RUNG wire#powerrail
      Contact( #BR07wAlm2.%X2 )
      Contact( #BR07wAlm2.%X3 )
      wire#w1
      Coil( "BMS2".BR07xSSFltSt )
   END_RUNG
   RUNG wire#powerrail
      Contact( #BR07wAlm3.%X6 )
   END_RUNG wire#w1
   // the same network as SCL:
   "BMS2".BR07xSSFltSt := (#BR07wAlm2.%X2 AND #BR07wAlm2.%X3) OR #BR07wAlm3.%X6;
END_REGION

REGION Network 90: BMS2 BR07 Fault
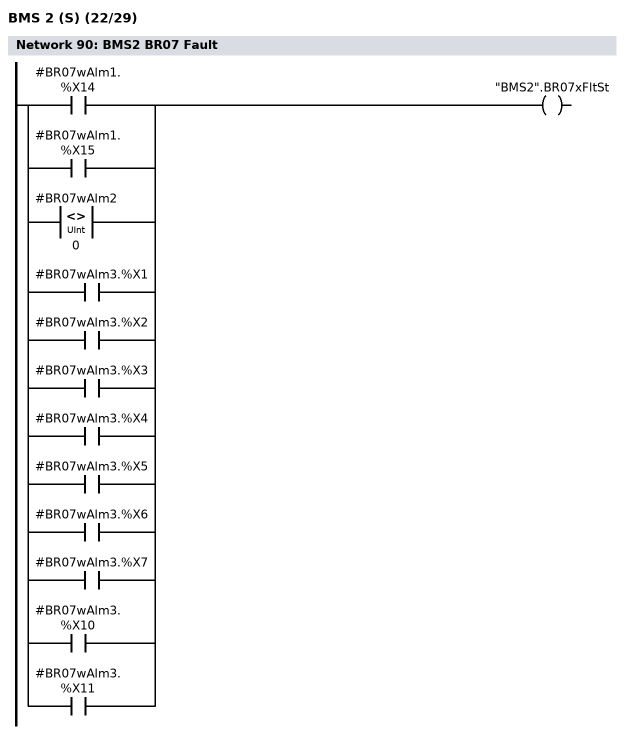
   RUNG wire#powerrail
      Contact( #BR07wAlm1.%X14 )
      wire#w1
      Coil( "BMS2".BR07xFltSt )
   END_RUNG
   RUNG wire#powerrail
      Contact( #BR07wAlm1.%X15 )
   END_RUNG wire#w1
   RUNG wire#powerrail
      { S7_Templates := "SrcType := UInt" } NE_Contact(in1 := #BR07wAlm2, in2 := 0)
   END_RUNG wire#w1
   RUNG wire#powerrail
      Contact( #BR07wAlm3.%X1 )
   END_RUNG wire#w1
   RUNG wire#powerrail
      Contact( #BR07wAlm3.%X2 )
   END_RUNG wire#w1
   RUNG wire#powerrail
      Contact( #BR07wAlm3.%X3 )
   END_RUNG wire#w1
   RUNG wire#powerrail
      Contact( #BR07wAlm3.%X4 )
   END_RUNG wire#w1
   RUNG wire#powerrail
      Contact( #BR07wAlm3.%X5 )
   END_RUNG wire#w1
   RUNG wire#powerrail
      Contact( #BR07wAlm3.%X6 )
   END_RUNG wire#w1
   RUNG wire#powerrail
      Contact( #BR07wAlm3.%X7 )
   END_RUNG wire#w1
   RUNG wire#powerrail
      Contact( #BR07wAlm3.%X10 )
   END_RUNG wire#w1
   RUNG wire#powerrail
      Contact( #BR07wAlm3.%X11 )
   END_RUNG wire#w1
   // the same network as SCL:
   "BMS2".BR07xFltSt := #BR07wAlm1.%X14 OR #BR07wAlm1.%X15 OR (#BR07wAlm2 <> 0) OR #BR07wAlm3.%X1 OR #BR07wAlm3.%X2 OR #BR07wAlm3.%X3 OR #BR07wAlm3.%X4 OR #BR07wAlm3.%X5 OR #BR07wAlm3.%X6 OR #BR07wAlm3.%X7 OR #BR07wAlm3.%X10 OR #BR07wAlm3.%X11;
END_REGION

REGION Network 91: BMS2 BR07 Alarm
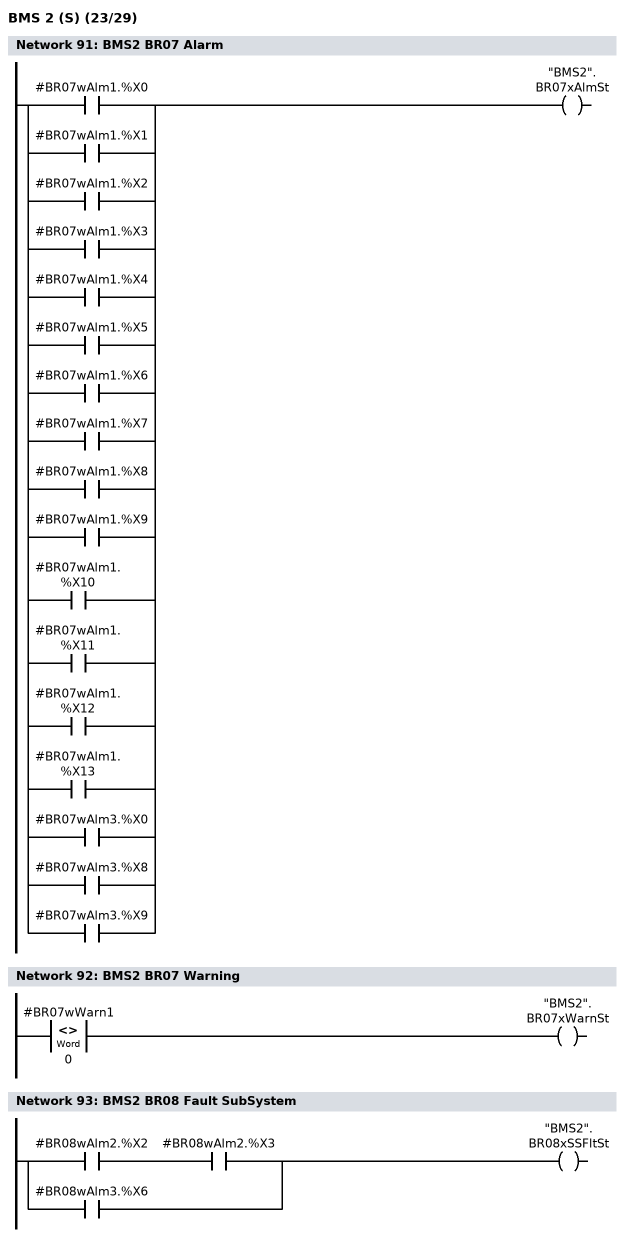
   RUNG wire#powerrail
      Contact( #BR07wAlm1.%X0 )
      wire#w1
      Coil( "BMS2".BR07xAlmSt )
   END_RUNG
   RUNG wire#powerrail
      Contact( #BR07wAlm1.%X1 )
   END_RUNG wire#w1
   RUNG wire#powerrail
      Contact( #BR07wAlm1.%X2 )
   END_RUNG wire#w1
   RUNG wire#powerrail
      Contact( #BR07wAlm1.%X3 )
   END_RUNG wire#w1
   RUNG wire#powerrail
      Contact( #BR07wAlm1.%X4 )
   END_RUNG wire#w1
   RUNG wire#powerrail
      Contact( #BR07wAlm1.%X5 )
   END_RUNG wire#w1
   RUNG wire#powerrail
      Contact( #BR07wAlm1.%X6 )
   END_RUNG wire#w1
   RUNG wire#powerrail
      Contact( #BR07wAlm1.%X7 )
   END_RUNG wire#w1
   RUNG wire#powerrail
      Contact( #BR07wAlm1.%X8 )
   END_RUNG wire#w1
   RUNG wire#powerrail
      Contact( #BR07wAlm1.%X9 )
   END_RUNG wire#w1
   RUNG wire#powerrail
      Contact( #BR07wAlm1.%X10 )
   END_RUNG wire#w1
   RUNG wire#powerrail
      Contact( #BR07wAlm1.%X11 )
   END_RUNG wire#w1
   RUNG wire#powerrail
      Contact( #BR07wAlm1.%X12 )
   END_RUNG wire#w1
   RUNG wire#powerrail
      Contact( #BR07wAlm1.%X13 )
   END_RUNG wire#w1
   RUNG wire#powerrail
      Contact( #BR07wAlm3.%X0 )
   END_RUNG wire#w1
   RUNG wire#powerrail
      Contact( #BR07wAlm3.%X8 )
   END_RUNG wire#w1
   RUNG wire#powerrail
      Contact( #BR07wAlm3.%X9 )
   END_RUNG wire#w1
   // the same network as SCL:
   "BMS2".BR07xAlmSt := #BR07wAlm1.%X0 OR #BR07wAlm1.%X1 OR #BR07wAlm1.%X2 OR #BR07wAlm1.%X3 OR #BR07wAlm1.%X4 OR #BR07wAlm1.%X5 OR #BR07wAlm1.%X6 OR #BR07wAlm1.%X7 OR #BR07wAlm1.%X8 OR #BR07wAlm1.%X9 OR #BR07wAlm1.%X10 OR #BR07wAlm1.%X11 OR #BR07wAlm1.%X12 OR #BR07wAlm1.%X13 OR #BR07wAlm3.%X0 OR #BR07wAlm3.%X8 OR #BR07wAlm3.%X9;
END_REGION

REGION Network 92: BMS2 BR07 Warning
   RUNG wire#powerrail
      { S7_Templates := "SrcType := Word" } NE_Contact(in1 := #BR07wWarn1, in2 := 0)
      Coil( "BMS2".BR07xWarnSt )
   END_RUNG
   // the same network as SCL:
   "BMS2".BR07xWarnSt := #BR07wWarn1 <> 0;
END_REGION

REGION Network 93: BMS2 BR08 Fault SubSystem
   RUNG wire#powerrail
      Contact( #BR08wAlm2.%X2 )
      Contact( #BR08wAlm2.%X3 )
      wire#w1
      Coil( "BMS2".BR08xSSFltSt )
   END_RUNG
   RUNG wire#powerrail
      Contact( #BR08wAlm3.%X6 )
   END_RUNG wire#w1
   // the same network as SCL:
   "BMS2".BR08xSSFltSt := (#BR08wAlm2.%X2 AND #BR08wAlm2.%X3) OR #BR08wAlm3.%X6;
END_REGION

REGION Network 94: BMS2 BR08 Fault
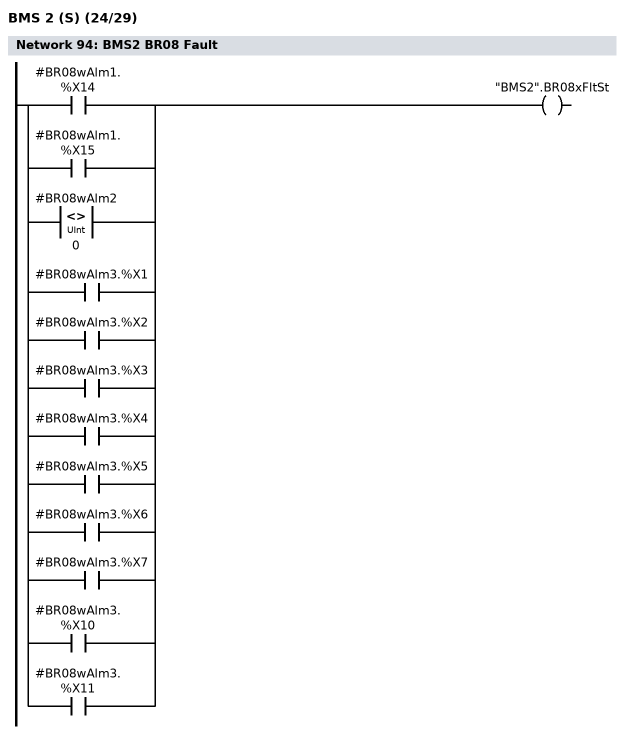
   RUNG wire#powerrail
      Contact( #BR08wAlm1.%X14 )
      wire#w1
      Coil( "BMS2".BR08xFltSt )
   END_RUNG
   RUNG wire#powerrail
      Contact( #BR08wAlm1.%X15 )
   END_RUNG wire#w1
   RUNG wire#powerrail
      { S7_Templates := "SrcType := UInt" } NE_Contact(in1 := #BR08wAlm2, in2 := 0)
   END_RUNG wire#w1
   RUNG wire#powerrail
      Contact( #BR08wAlm3.%X1 )
   END_RUNG wire#w1
   RUNG wire#powerrail
      Contact( #BR08wAlm3.%X2 )
   END_RUNG wire#w1
   RUNG wire#powerrail
      Contact( #BR08wAlm3.%X3 )
   END_RUNG wire#w1
   RUNG wire#powerrail
      Contact( #BR08wAlm3.%X4 )
   END_RUNG wire#w1
   RUNG wire#powerrail
      Contact( #BR08wAlm3.%X5 )
   END_RUNG wire#w1
   RUNG wire#powerrail
      Contact( #BR08wAlm3.%X6 )
   END_RUNG wire#w1
   RUNG wire#powerrail
      Contact( #BR08wAlm3.%X7 )
   END_RUNG wire#w1
   RUNG wire#powerrail
      Contact( #BR08wAlm3.%X10 )
   END_RUNG wire#w1
   RUNG wire#powerrail
      Contact( #BR08wAlm3.%X11 )
   END_RUNG wire#w1
   // the same network as SCL:
   "BMS2".BR08xFltSt := #BR08wAlm1.%X14 OR #BR08wAlm1.%X15 OR (#BR08wAlm2 <> 0) OR #BR08wAlm3.%X1 OR #BR08wAlm3.%X2 OR #BR08wAlm3.%X3 OR #BR08wAlm3.%X4 OR #BR08wAlm3.%X5 OR #BR08wAlm3.%X6 OR #BR08wAlm3.%X7 OR #BR08wAlm3.%X10 OR #BR08wAlm3.%X11;
END_REGION

REGION Network 95: BMS2 BR08 Alarm
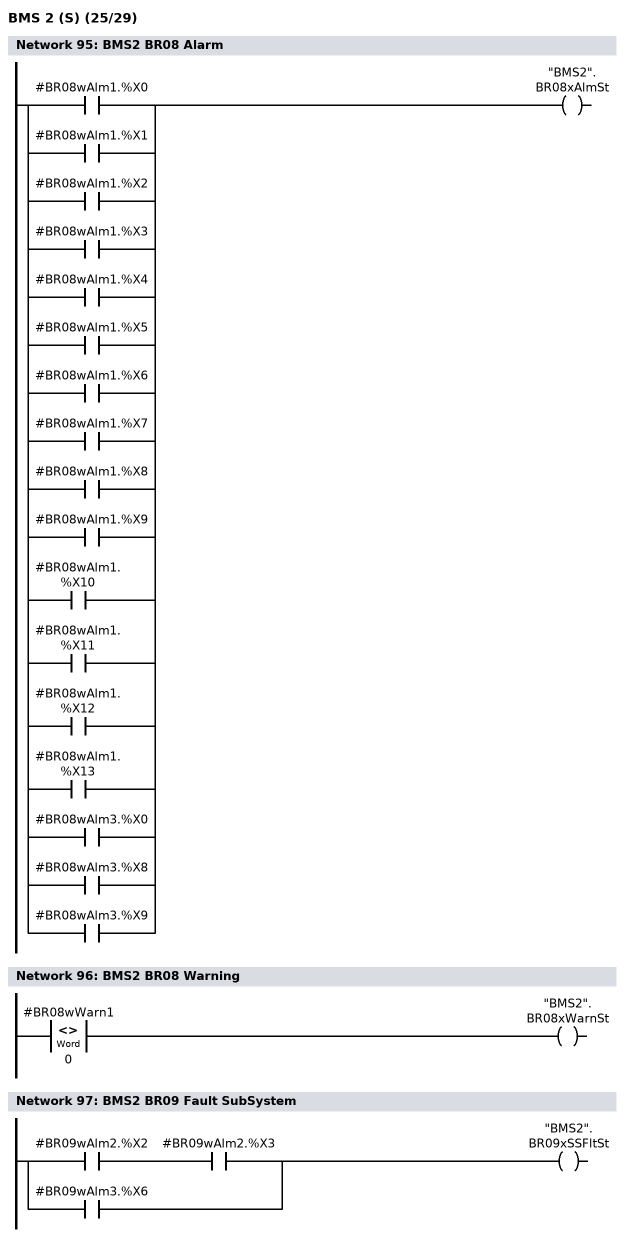
   RUNG wire#powerrail
      Contact( #BR08wAlm1.%X0 )
      wire#w1
      Coil( "BMS2".BR08xAlmSt )
   END_RUNG
   RUNG wire#powerrail
      Contact( #BR08wAlm1.%X1 )
   END_RUNG wire#w1
   RUNG wire#powerrail
      Contact( #BR08wAlm1.%X2 )
   END_RUNG wire#w1
   RUNG wire#powerrail
      Contact( #BR08wAlm1.%X3 )
   END_RUNG wire#w1
   RUNG wire#powerrail
      Contact( #BR08wAlm1.%X4 )
   END_RUNG wire#w1
   RUNG wire#powerrail
      Contact( #BR08wAlm1.%X5 )
   END_RUNG wire#w1
   RUNG wire#powerrail
      Contact( #BR08wAlm1.%X6 )
   END_RUNG wire#w1
   RUNG wire#powerrail
      Contact( #BR08wAlm1.%X7 )
   END_RUNG wire#w1
   RUNG wire#powerrail
      Contact( #BR08wAlm1.%X8 )
   END_RUNG wire#w1
   RUNG wire#powerrail
      Contact( #BR08wAlm1.%X9 )
   END_RUNG wire#w1
   RUNG wire#powerrail
      Contact( #BR08wAlm1.%X10 )
   END_RUNG wire#w1
   RUNG wire#powerrail
      Contact( #BR08wAlm1.%X11 )
   END_RUNG wire#w1
   RUNG wire#powerrail
      Contact( #BR08wAlm1.%X12 )
   END_RUNG wire#w1
   RUNG wire#powerrail
      Contact( #BR08wAlm1.%X13 )
   END_RUNG wire#w1
   RUNG wire#powerrail
      Contact( #BR08wAlm3.%X0 )
   END_RUNG wire#w1
   RUNG wire#powerrail
      Contact( #BR08wAlm3.%X8 )
   END_RUNG wire#w1
   RUNG wire#powerrail
      Contact( #BR08wAlm3.%X9 )
   END_RUNG wire#w1
   // the same network as SCL:
   "BMS2".BR08xAlmSt := #BR08wAlm1.%X0 OR #BR08wAlm1.%X1 OR #BR08wAlm1.%X2 OR #BR08wAlm1.%X3 OR #BR08wAlm1.%X4 OR #BR08wAlm1.%X5 OR #BR08wAlm1.%X6 OR #BR08wAlm1.%X7 OR #BR08wAlm1.%X8 OR #BR08wAlm1.%X9 OR #BR08wAlm1.%X10 OR #BR08wAlm1.%X11 OR #BR08wAlm1.%X12 OR #BR08wAlm1.%X13 OR #BR08wAlm3.%X0 OR #BR08wAlm3.%X8 OR #BR08wAlm3.%X9;
END_REGION

REGION Network 96: BMS2 BR08 Warning
   RUNG wire#powerrail
      { S7_Templates := "SrcType := Word" } NE_Contact(in1 := #BR08wWarn1, in2 := 0)
      Coil( "BMS2".BR08xWarnSt )
   END_RUNG
   // the same network as SCL:
   "BMS2".BR08xWarnSt := #BR08wWarn1 <> 0;
END_REGION

REGION Network 97: BMS2 BR09 Fault SubSystem
   RUNG wire#powerrail
      Contact( #BR09wAlm2.%X2 )
      Contact( #BR09wAlm2.%X3 )
      wire#w1
      Coil( "BMS2".BR09xSSFltSt )
   END_RUNG
   RUNG wire#powerrail
      Contact( #BR09wAlm3.%X6 )
   END_RUNG wire#w1
   // the same network as SCL:
   "BMS2".BR09xSSFltSt := (#BR09wAlm2.%X2 AND #BR09wAlm2.%X3) OR #BR09wAlm3.%X6;
END_REGION

REGION Network 98: BMS2 BR09 Fault
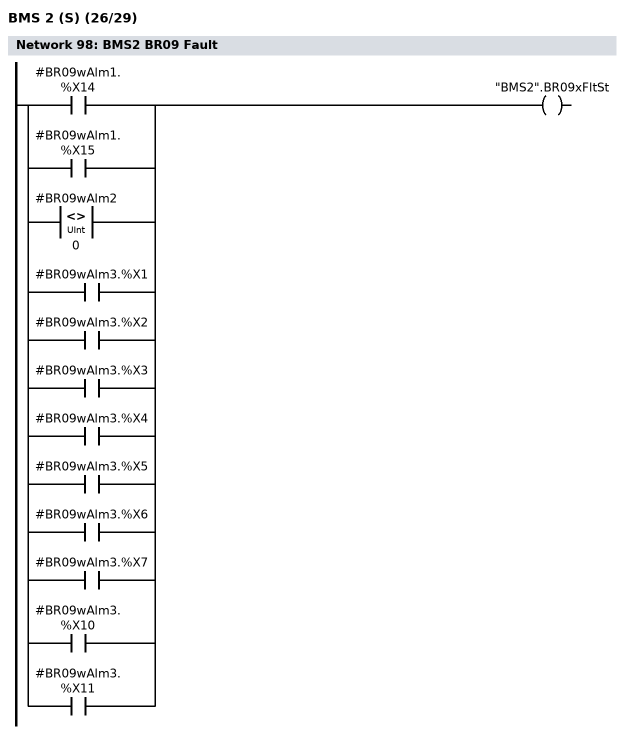
   RUNG wire#powerrail
      Contact( #BR09wAlm1.%X14 )
      wire#w1
      Coil( "BMS2".BR09xFltSt )
   END_RUNG
   RUNG wire#powerrail
      Contact( #BR09wAlm1.%X15 )
   END_RUNG wire#w1
   RUNG wire#powerrail
      { S7_Templates := "SrcType := UInt" } NE_Contact(in1 := #BR09wAlm2, in2 := 0)
   END_RUNG wire#w1
   RUNG wire#powerrail
      Contact( #BR09wAlm3.%X1 )
   END_RUNG wire#w1
   RUNG wire#powerrail
      Contact( #BR09wAlm3.%X2 )
   END_RUNG wire#w1
   RUNG wire#powerrail
      Contact( #BR09wAlm3.%X3 )
   END_RUNG wire#w1
   RUNG wire#powerrail
      Contact( #BR09wAlm3.%X4 )
   END_RUNG wire#w1
   RUNG wire#powerrail
      Contact( #BR09wAlm3.%X5 )
   END_RUNG wire#w1
   RUNG wire#powerrail
      Contact( #BR09wAlm3.%X6 )
   END_RUNG wire#w1
   RUNG wire#powerrail
      Contact( #BR09wAlm3.%X7 )
   END_RUNG wire#w1
   RUNG wire#powerrail
      Contact( #BR09wAlm3.%X10 )
   END_RUNG wire#w1
   RUNG wire#powerrail
      Contact( #BR09wAlm3.%X11 )
   END_RUNG wire#w1
   // the same network as SCL:
   "BMS2".BR09xFltSt := #BR09wAlm1.%X14 OR #BR09wAlm1.%X15 OR (#BR09wAlm2 <> 0) OR #BR09wAlm3.%X1 OR #BR09wAlm3.%X2 OR #BR09wAlm3.%X3 OR #BR09wAlm3.%X4 OR #BR09wAlm3.%X5 OR #BR09wAlm3.%X6 OR #BR09wAlm3.%X7 OR #BR09wAlm3.%X10 OR #BR09wAlm3.%X11;
END_REGION

REGION Network 99: BMS2 BR09 Alarm
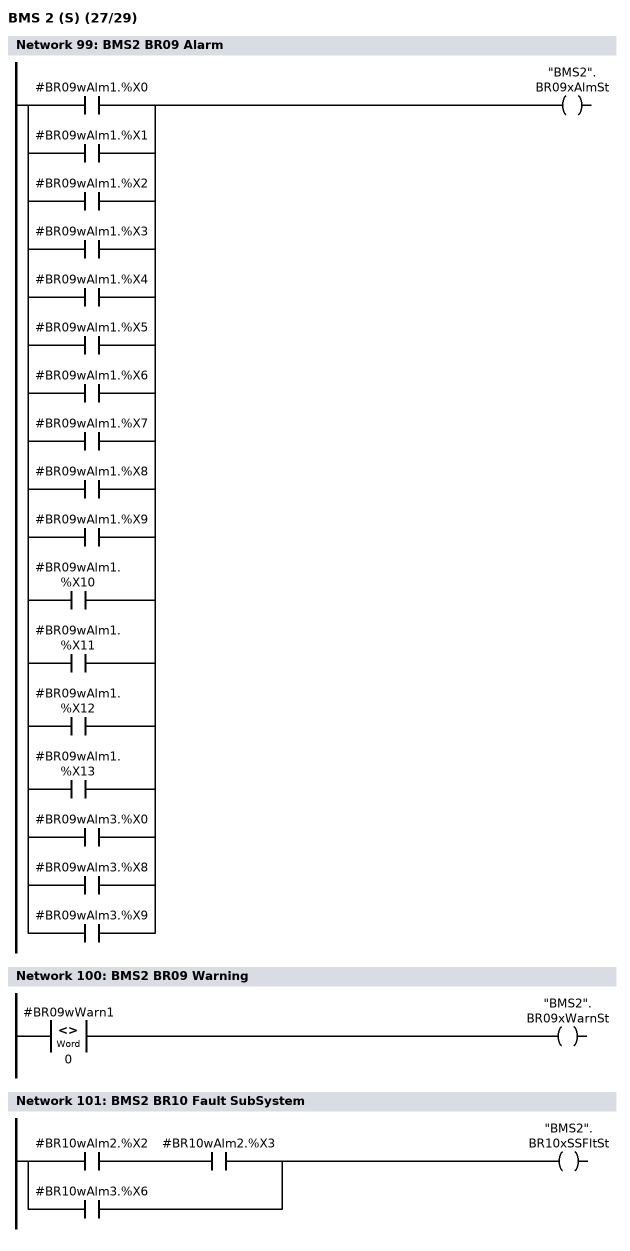
   RUNG wire#powerrail
      Contact( #BR09wAlm1.%X0 )
      wire#w1
      Coil( "BMS2".BR09xAlmSt )
   END_RUNG
   RUNG wire#powerrail
      Contact( #BR09wAlm1.%X1 )
   END_RUNG wire#w1
   RUNG wire#powerrail
      Contact( #BR09wAlm1.%X2 )
   END_RUNG wire#w1
   RUNG wire#powerrail
      Contact( #BR09wAlm1.%X3 )
   END_RUNG wire#w1
   RUNG wire#powerrail
      Contact( #BR09wAlm1.%X4 )
   END_RUNG wire#w1
   RUNG wire#powerrail
      Contact( #BR09wAlm1.%X5 )
   END_RUNG wire#w1
   RUNG wire#powerrail
      Contact( #BR09wAlm1.%X6 )
   END_RUNG wire#w1
   RUNG wire#powerrail
      Contact( #BR09wAlm1.%X7 )
   END_RUNG wire#w1
   RUNG wire#powerrail
      Contact( #BR09wAlm1.%X8 )
   END_RUNG wire#w1
   RUNG wire#powerrail
      Contact( #BR09wAlm1.%X9 )
   END_RUNG wire#w1
   RUNG wire#powerrail
      Contact( #BR09wAlm1.%X10 )
   END_RUNG wire#w1
   RUNG wire#powerrail
      Contact( #BR09wAlm1.%X11 )
   END_RUNG wire#w1
   RUNG wire#powerrail
      Contact( #BR09wAlm1.%X12 )
   END_RUNG wire#w1
   RUNG wire#powerrail
      Contact( #BR09wAlm1.%X13 )
   END_RUNG wire#w1
   RUNG wire#powerrail
      Contact( #BR09wAlm3.%X0 )
   END_RUNG wire#w1
   RUNG wire#powerrail
      Contact( #BR09wAlm3.%X8 )
   END_RUNG wire#w1
   RUNG wire#powerrail
      Contact( #BR09wAlm3.%X9 )
   END_RUNG wire#w1
   // the same network as SCL:
   "BMS2".BR09xAlmSt := #BR09wAlm1.%X0 OR #BR09wAlm1.%X1 OR #BR09wAlm1.%X2 OR #BR09wAlm1.%X3 OR #BR09wAlm1.%X4 OR #BR09wAlm1.%X5 OR #BR09wAlm1.%X6 OR #BR09wAlm1.%X7 OR #BR09wAlm1.%X8 OR #BR09wAlm1.%X9 OR #BR09wAlm1.%X10 OR #BR09wAlm1.%X11 OR #BR09wAlm1.%X12 OR #BR09wAlm1.%X13 OR #BR09wAlm3.%X0 OR #BR09wAlm3.%X8 OR #BR09wAlm3.%X9;
END_REGION

REGION Network 100: BMS2 BR09 Warning
   RUNG wire#powerrail
      { S7_Templates := "SrcType := Word" } NE_Contact(in1 := #BR09wWarn1, in2 := 0)
      Coil( "BMS2".BR09xWarnSt )
   END_RUNG
   // the same network as SCL:
   "BMS2".BR09xWarnSt := #BR09wWarn1 <> 0;
END_REGION

REGION Network 101: BMS2 BR10 Fault SubSystem
   RUNG wire#powerrail
      Contact( #BR10wAlm2.%X2 )
      Contact( #BR10wAlm2.%X3 )
      wire#w1
      Coil( "BMS2".BR10xSSFltSt )
   END_RUNG
   RUNG wire#powerrail
      Contact( #BR10wAlm3.%X6 )
   END_RUNG wire#w1
   // the same network as SCL:
   "BMS2".BR10xSSFltSt := (#BR10wAlm2.%X2 AND #BR10wAlm2.%X3) OR #BR10wAlm3.%X6;
END_REGION

REGION Network 102: BMS2 BR10 Fault
